(* IEC 61131-3 sources: beebread/doc (part 7) *)

(* ---------------------------------------------- *)
C_SND:
	IF S_BUF.SIZE > 0 THEN
		IF c_ready AND c_enable THEN
			IF NOT s_active THEN
				s_total := LIMIT(0,UINT_TO_INT(S_BUF.SIZE),r_max_size); (* limit and pass total number of bytes *)
				s_cur_pos  := 0;
				s_cur_size := 0;
				s_active := TRUE; (* activate send mode *)
			END_IF;

			s_cur_pos := s_cur_pos + s_cur_size; (* determine new send data position *)
			IF s_total > s_cur_pos THEN (* more data to send? *)
				s_cur_size := s_total - s_cur_pos;
				s_cur_size := LIMIT(0, s_cur_size, s_max_size); (* limit telegram length *)
				s_time := tx; (* reset send timer *)
				r_time := tx; (* reset receive timer *)
				state := C_SND_WAIT1;
			ELSE (* no more send data -> stop sending *)
				s_active := FALSE;
				S_BUF.SIZE := 0;
				state := C_WAIT;
			END_IF;
		END_IF;
	END_IF;

C_SND_WAIT1:
	IF udp_mode THEN
		fbSendTo(bExecute := FALSE );
		fbSendTo(bExecute := TRUE, sSrvNetId := sSrvNetId, hSocket := socket , cbLen := s_cur_size, pSrc := REF(S_BUF.BUFFER[s_cur_pos]), sRemoteHost := s_ip_str, nRemotePort := c_port, tTimeout:= TIME_OUT);
		fbSendTo.bExecute := FALSE;
	ELSE
		fbSend(bExecute := FALSE);
		fbSend(bExecute := TRUE, sSrvNetId := sSrvNetId, hSocket := socket , cbLen:= s_cur_size, pSrc:=REF(S_BUF.BUFFER[s_cur_pos]), tTimeout:= TIME_OUT);
		fbSend.bExecute := FALSE;
	END_IF;
	state := C_SND_WAIT2;

C_SND_WAIT2:
	IF udp_mode THEN
		fbSendTo();
		Send_Busy := fbSendTo.bBusy;
		Send_Error := fbSendTo.bError;
		Send_ErrId := fbSendTo.nErrId;
	ELSE
		fbSend();
		Send_Busy := fbSend.bBusy;
		Send_Error := fbSend.bError;
		Send_ErrId := fbSend.nErrId;
	END_IF;

	IF NOT Send_Busy THEN
		IF NOT Send_Error THEN
    			(*####################  DEBUG-MESSAGE  ###################################*)
			(*########################################################################*)
			state := C_SND;
		ELSE
			nErrId := Send_ErrId;
			state := C_WAIT;
    			(*####################  DEBUG-MESSAGE  ###################################*)
			(*########################################################################*)
		END_IF;
	END_IF;

END_CASE;

(* ---------------------------------------------- *)

IF c_ready THEN
	IF NOT c_ready_old THEN (* connection established - rising edge detected *)
		IP_C.C_STATE := 254;
		IP_C.TIME_RESET := TRUE; (* reset all timers *)
    		(*####################  DEBUG-MESSAGE  ###################################*)
		(*########################################################################*)
	ELSE
		IP_C.C_STATE := 255; (* connection is established *)
	END_IF;
ELSE
	IF c_ready_old THEN (* connection closed - falling edge detected *)
		IP_C.C_STATE := 1;
		IP_C.MAILBOX[1] := 0; (* reset receive info *)
		IP_C.MAILBOX[2] := 0; (* reset send pause *)
		IP_C.MAILBOX[3] := 0; (* reset receive pause *)
		IF NOT new_connection THEN
			s_active := FALSE; (* stop send activities *)
			S_BUF.SIZE := 0; (* clear send length *)
			(*IP_C.TIME_RESET := TRUE; *) (* reset all timers *)
		END_IF;
    		(*####################  DEBUG-MESSAGE  ###################################*)
		(*########################################################################*)

	ELSE
		IP_C.C_STATE := 0; (* connection is closed *)
	END_IF;
END_IF;

c_ready_old := c_ready;

(* ---------------------------------------------- *)

IF IP_C.R_OBSERVE = FALSE OR s_active THEN
    r_time := tx;
END_IF;

IF c_status = 0 AND tx - c_time > error_time AND c_enable AND NOT c_ready AND c_mode < 2 THEN (* Connect Timeout *)
	c_status := 255; (* output timeout error *)
END_IF;
IF s_status = 0 AND tx - s_time > error_time AND s_active THEN (* Send Timeout *)
	s_status := 255; (* output timeout error *)
END_IF;
IF r_status = 0 AND tx - r_time > error_time AND c_ready AND IP_C.R_OBSERVE THEN (* Receive Timeout *)
	r_status := 255; (* output timeout error *)
END_IF;

IP_C.ERROR := DWORD_OF_BYTE(c_status,s_status,r_status,0);

(*####################  DEBUG-MESSAGE  ###################################*)
(*########################################################################*)
END_FUNCTION_BLOCK

FUNCTION_BLOCK IP_CONTROL2
VAR_IN_OUT
	IP_C : IP_C; (* IP_Control management structure *)
	S_BUF : NETWORK_BUFFER_SHORT; (* external send buffer *)
	R_BUF : NETWORK_BUFFER_SHORT; (* external receive buffer *)
END_VAR
VAR_INPUT
	IP : DWORD; (* IP address *)
	PORT : WORD; (* port number *)
	TIME_OUT : TIME; (* monitoring time connect / send / receive *)
END_VAR
VAR
	c_time : UDINT; (* CONNECT time (time without a connection) *)
	s_time : UDINT; (* SEND time    (time since last data sent) *)
	r_time : UDINT; (* RECEIVE time (time since last data received) *)

	c_enable : BOOL; (* Connect: enable *)
	c_ip : DWORD; (* Connect: current IP address *)
	c_ip_str : STRING(15);
	c_port : WORD; (* Connect: current port number *)
	c_mode : BYTE; (* Connect: current mode UDP/TCP...... *)
	c_status : BYTE; (* Connect: Status (Errorcode) *)
	c_ready : BOOL; (* Connect: connection established *)
	c_ready_old : BOOL; (* Connect: last state of c_ready for edge evaluation *)

	s_total : INT; (* Send: total number of bytes to send *)
	s_cur_pos : INT; (* Send: current send position *)
	s_cur_size : INT; (* Send: current send size *)
	s_max_size : INT; (* Send: maximum telegram length for sending *)
	s_active : BOOL; (* Send: data sending is active *)
	s_status : BYTE; (* Send: Status (Errorcodes) *)
	s_ip_str : STRING(15);
	s_ip_exist : BOOL;

	r_status : BYTE; (* Receive: Status (Errorcodes) *)
	r_count : INT; (* Receive: number of received bytes *)
	r_offset : INT; (* Receive: current position in external receive buffer *)
	r_max_size : INT; (* Receive: size of the external receive buffer*)

	new_connection : BOOL; (* new connection parameters available *)
	tx : DWORD; (* last time value *)
	error_time : DWORD; (* current timeout value *)

	state: BYTE; (* step flag for connect *)
	bytes_received : DINT;
	udp_mode : BOOL;

	socket : T_HSOCKET;
	server : T_HSOCKET;
	fbCreate	: FB_SocketUdpCreate;
	fbConnect : FB_SocketConnect;
	fbClose : FB_SocketClose;
	fbSendTo : FB_SocketUdpSendTo;
	fbReceiveFrom : FB_SocketUdpReceiveFrom;
	fbSend : FB_SocketSend;
	fbReceive : FB_SocketReceive;
	fbListen : FB_SocketListen;
	fbAccept : FB_SocketAccept;
	nErrId : UDINT;
	Send_Busy : BOOL;
	Send_Error : BOOL;
	Send_ErrId : UDINT;

	IPCR : IP_CONTROL_RESET;

END_VAR

VAR CONSTANT
	STOP : BYTE := 0;
	UDP_INIT : BYTE:= 31;
	UDP_INIT_WAIT : BYTE:= 32;
	TC_INIT : BYTE := 51;
	TC_CONNECT : BYTE:= 52;
	TS_INIT : BYTE:= 53;
	TS_LISTEN_WAIT : BYTE:= 54;
	TS_ACCEPT : BYTE:= 55;
	TS_ACCEPT_WAIT : BYTE:= 56;
	C_CLOSE : BYTE := 190;
	C_CLOSE_WAIT : BYTE:= 191;
	C_CLOSE2 : BYTE := 192;
	C_CLOSE_WAIT2 : BYTE:= 193;
	C_WAIT : BYTE := 200;
	C_REC : BYTE := 210;
	C_REC_WAIT : BYTE := 211;
	C_SND : BYTE := 220;
	C_SND_WAIT1 : BYTE := 221;
	C_SND_WAIT2 : BYTE := 222;
END_VAR

(* on PLC reset or program download all old connections are closed *)
IPCR();
IF NOT IPCR.READY THEN RETURN; END_IF;

(* ---------------------- Debug-Message ----------------------------*)
(* -----------------------------------------------------------------------------*)

(* read system time *)
tx := T_PLC_MS();

IF IP_C.C_PORT = 0 THEN
	IP_C.C_PORT := PORT; (* replace the given PORT with the configured PORT *)
END_IF;
IF IP_C.C_IP = 0 AND IP_C.C_MODE < 4 THEN
	IP_C.C_IP := IP; (* replace the given IP with the configured IP *)
END_IF;

new_connection := c_ip <> IP_C.C_IP OR c_mode <> IP_C.C_MODE OR c_port <> IP_C.C_PORT; (* new connection requested? *)
c_enable := IP_C.C_ENABLE AND NOT new_connection;

IF IP_C.C_ENABLE AND IP_C.ERROR = 0 AND state = STOP THEN (* enabled, no error, no socket open *)
	c_ip   := IP_C.C_IP;
	c_mode := IP_C.C_MODE;
	c_port := IP_C.C_PORT;
	c_ip_str := IP4_TO_STRING(c_ip);
	udp_mode := C_MODE.0; (* Mode 1,3,5 = udp *)

	error_time := TIME_TO_DWORD(MAX(T#200ms,TIME_OUT));
	IP_C.TIME_RESET := TRUE; (* reset all timers *)
	r_max_size := SIZEOF(R_BUF.BUFFER);
	s_max_size := SIZEOF(S_BUF.BUFFER);

	IF udp_mode THEN (* Mode: 1,3,5 = UDP CLIENT/SERVER *)
		state := UDP_INIT;
	ELSIF c_mode = 0 THEN (* Mode: 0 = TCP CLIENT *)
		state := TC_INIT;
	ELSE
		state := TS_INIT; (* Mode: 2,4 = TCP SERVER *)
	END_IF;

	IF c_mode < 5 THEN (* set receiver IP *)
		s_ip_str := c_ip_str;
		s_ip_exist := TRUE;
	ELSE
		s_ip_str := '';
		s_ip_exist := FALSE;
	END_IF;

	(* ---------------------- Debug-Message ----------------------------*)
	(* -----------------------------------------------------------------------------*)

END_IF;

(* ---------------------- Debug-Message ----------------------------*)
(* -----------------------------------------------------------------------------*)

IF IP_C.TIME_RESET THEN (* reset all timers *)
	IP_C.TIME_RESET := FALSE; (* clear reset *)
	c_time := tx; (* reset connect timer *)
	s_time := tx; (* reset send timer *)
	r_time := tx; (* reset receive timer *)

	c_status := BYTE#0; (* reset last connect error *)
	s_status := BYTE#0; (* reset last send error *)
	r_status := BYTE#0; (* reset last receive error *)
END_IF;

(* ---------------------------------------------- *)

CASE state OF

UDP_INIT: (* UDP_CLIENT + SERVER *)

	fbCreate(bExecute := FALSE);
	fbCreate(	bExecute := TRUE , sSrvNetId := sSrvNetId, sLocalHost := sLocalHost, nLocalPort := SEL(c_mode = 1,c_port,0) , tTimeOut := TIME_OUT);
	fbCreate.bExecute := FALSE; (* presetting *)
	state := UDP_INIT_WAIT;

UDP_INIT_WAIT:
	fbCreate();
	IF NOT fbCreate.bBusy THEN
		IF NOT fbCreate.bError THEN
			socket := fbCreate.hSocket;
			c_ready := TRUE; (* Connected *)
			state := C_WAIT;
		ELSE
			c_status := 1; (* FB_SocketUdpCreate failed *)
			nErrId := fbCreate.nErrId;
			state := C_CLOSE;
		END_IF;
	END_IF;

(* ---------------------------------------------- *)
TC_INIT: (* TCP CLIENT (ACTIVE) *)
	fbConnect(bExecute := FALSE);
	fbConnect(bExecute := TRUE, sSrvNetId := sSrvNetId, sRemoteHost := c_ip_str, nRemotePort := c_port, tTimeout := TIME_OUT);
	fbConnect.bExecute := FALSE; (* presetting *)
	state := TC_CONNECT;

(* ---------------------------------------------- *)
TC_CONNECT:
	IF NOT c_enable OR c_status = 255 THEN (* not enabled or connect timeout *)
		state := C_CLOSE;
	END_IF;

	fbConnect();
	IF NOT fbConnect.bBusy THEN
		IF fbConnect.bError THEN
			nErrID := fbConnect.nErrId;
			state :=TC_INIT; (* try again *)
		ELSE
			socket := fbConnect.hSocket;
			c_ready := TRUE; (* Connected *)
			state := C_WAIT;
		END_IF;
	END_IF;
(* ---------------------------------------------- *)
TS_INIT: (* TCP SERVER (PASSIVE) *)
	fbListen(bExecute := FALSE);
	fbListen(bExecute := TRUE , sSrvNetId:= sSrvNetId , sLocalHost:= sLocalHost , nLocalPort:= c_port , tTimeout:= TIME_OUT);
	fbListen.bExecute := FALSE;
	state := TS_LISTEN_WAIT;
(* ---------------------------------------------- *)
TS_LISTEN_WAIT:
	fbListen();
	IF NOT fbListen.bBusy THEN
		IF fbListen.bError THEN
			c_status := 3; (* FB_SocketListen failed *)
			nErrID := fbListen.nErrId;
			state := C_CLOSE;
		ELSE
			server := fbListen.hListener;
			state := TS_ACCEPT;
		END_IF;
	END_IF;
(* ---------------------------------------------- *)
TS_ACCEPT:
	fbAccept(bExecute := FALSE);
	fbAccept(bExecute := TRUE, sSrvNetId := sSrvNetId, hListener := server, tTimeout := TIME_OUT);
	fbAccept.bExecute := FALSE;
	state := TS_ACCEPT_WAIT;
(* ---------------------------------------------- *)
TS_ACCEPT_WAIT:
	fbAccept();
	IF NOT fbAccept.bBusy THEN

		state := TS_ACCEPT; (* presetting  *)

		IF fbAccept.bError THEN
			c_status := 4; (* FB_SocketAccept failed *)
			nErrID := fbAccept.nErrId;
			state := C_CLOSE;
		ELSE (* no error *)
			IF fbAccept.bAccepted THEN
				socket := fbAccept.hSocket;
				IF socket.remoteAddr.sAddr  <> c_ip_str AND c_mode <> 4 THEN
					state := C_CLOSE; (* reject remote - close connection *)
				ELSE
					state := C_WAIT;
					c_ready := TRUE; (* Connected *)
				END_IF;
			END_IF; (* fbAccept.bAccepted *)
		END_IF; (* NOT fbAccept.bError *)
	END_IF; (*  NOT fbAccept.bBusy *)
(* ---------------------------------------------- *)
C_CLOSE:
	c_ready := FALSE;
	IF socket.handle > 0 THEN
		fbClose(bExecute := FALSE );
		fbClose(bExecute := TRUE, sSrvNetId := sSrvNetId,	hSocket := socket);
		fbClose.bExecute := FALSE;
		state := C_CLOSE_WAIT;
	ELSE
		state:= C_CLOSE2;
	END_IF;

C_CLOSE_WAIT:
	fbClose();
	IF NOT fbClose.bBusy THEN
		socket := TCPADS_NULL_HSOCKET; (* reset socket *)
		nErrId:= SEL(fbClose.bError,0,fbClose.nErrId);
		state:= C_CLOSE2;
	END_IF;

C_CLOSE2:
	IF server.handle > 0 THEN
		fbClose(bExecute := FALSE );
		fbClose(bExecute := TRUE, sSrvNetId := sSrvNetId,	hSocket := server);
		fbClose.bExecute := FALSE;
		state := C_CLOSE_WAIT2;
	ELSE
		state:= STOP;
	END_IF;

C_CLOSE_WAIT2:
	fbClose();
	IF NOT fbClose.bBusy THEN
		server := TCPADS_NULL_HSOCKET; (* reset socket *)
		nErrId:= SEL(fbClose.bError,0,fbClose.nErrId);
		state:= STOP;
	END_IF;

(* ---------------------------------------------- *)

C_WAIT: (* wait for request to close *)
	IF NOT c_enable OR NOT c_ready THEN
		state:= C_CLOSE;
	ELSIF S_BUF.SIZE > 0 AND IP_C.MAILBOX[2] = 0 AND s_ip_exist THEN
		state:= C_SND;
	ELSIF IP_C.MAILBOX[3] = 0 THEN
		state:= C_REC;
	END_IF;

(* ---------------------------------------------- *)

C_REC: (* receive data *)
	IF R_BUF.SIZE >= INT_TO_UINT(r_max_size) THEN
		R_BUF.SIZE := UINT#0;
		r_status := 254; (* receive buffer reset due to overflow *)
	END_IF;

	r_offset := SEL(udp_mode,UINT_TO_INT(R_BUF.SIZE),0);
	r_count := r_max_size - r_offset;
	bytes_received := 0;

	IF udp_mode THEN
		fbReceiveFrom(bExecute := FALSE );
		fbReceiveFrom(bExecute:= TRUE, sSrvNetId := sSrvNetId, hSocket:= socket, cbLen := r_count, pDest:= REF(R_BUF.BUFFER), tTimeout:= TIME_OUT);
		fbReceiveFrom.bExecute := FALSE; (* presetting *)
	ELSE
		fbReceive(bExecute:= FALSE);
		fbReceive(bExecute:= TRUE, sSrvNetId := sSrvNetId , hSocket:= socket , cbLen:= r_count, pDest:= REF(R_BUF.BUFFER[r_offset]) , tTimeout:= TIME_OUT);
		fbReceive.bExecute:= FALSE;
	END_IF;
	state := C_REC_WAIT;

C_REC_WAIT:
	IF udp_mode THEN
		fbReceiveFrom(); (* UDP Mode *)
		IF NOT fbReceiveFrom.bBusy THEN
			IF NOT fbReceiveFrom.bError THEN
				IF fbReceiveFrom.nRecBytes > 0 THEN
					IF c_mode <> BYTE#5 AND fbReceiveFrom.sRemoteHost  <> c_ip_str THEN
						R_BUF.SIZE := UINT#0;
					ELSE
						bytes_received := fbReceiveFrom.nRecBytes;
						IF NOT s_ip_exist THEN
							s_ip_str := fbReceiveFrom.sRemoteHost;
							s_ip_exist := TRUE;
						END_IF;
					END_IF;
				END_IF;
				state := C_WAIT;
			ELSIF fbReceiveFrom.nErrId = 16#80072746 THEN (* connection closed by remote *)
				c_status := 253;
				c_ready := FALSE;
				state := C_WAIT;
			ELSE
				nErrId := fbReceiveFrom.nErrId;
				state := C_WAIT;
			END_IF;
		END_IF;
	ELSE
		fbReceive(); (* TCP Mode *)
		IF NOT fbReceive.bBusy THEN
			IF NOT fbReceive.bError THEN
				IF fbReceive.nRecBytes > 0 THEN
					bytes_received := fbReceive.nRecBytes;
				END_IF;
			ELSIF fbReceive.nErrId = 16#8004 THEN (* connection closed by remote *)
				c_status := 253;
				c_ready := FALSE;
			ELSE
				nErrId := fbReceive.nErrId;
			END_IF;
			state := C_WAIT;
		END_IF;
	END_IF;

	IF bytes_received > 0 THEN
		r_time := tx; (* reset receive timer *)
		R_BUF.SIZE := INT_TO_UINT(r_offset + DINT_TO_UINT(bytes_received)); (* enter current buffer size *)
		IP_C.MAILBOX[1] := IP_C.MAILBOX[1] + 1; (* Receive Info *)
		IF IP_C.MAILBOX[1] = 0 THEN IP_C.MAILBOX[1] := 1; END_IF;
		(* ---------------------- Debug-Message ----------------------------*)
		(* -----------------------------------------------------------------------------*)
	END_IF;

(* ---------------------------------------------- *)
C_SND:
	IF S_BUF.SIZE > 0 THEN
		IF c_ready AND c_enable THEN
			IF NOT s_active THEN
				s_total := LIMIT(0,UINT_TO_INT(S_BUF.SIZE),r_max_size); (* limit and pass total number of bytes *)
				s_cur_pos  := 0;
				s_cur_size := 0;
				s_active := TRUE; (* activate send mode *)
			END_IF;

			s_cur_pos := s_cur_pos + s_cur_size; (* determine new send data position *)
			IF s_total > s_cur_pos THEN (* more data to send? *)
				s_cur_size := s_total - s_cur_pos;
				s_cur_size := LIMIT(0, s_cur_size, s_max_size); (* limit telegram length *)
				s_time := tx; (* reset send timer *)
				r_time := tx; (* reset receive timer *)
				state := C_SND_WAIT1;
			ELSE (* no more send data -> stop sending *)
				s_active := FALSE;
				S_BUF.SIZE := 0;
				state := C_WAIT;
			END_IF;
		END_IF;
	END_IF;

C_SND_WAIT1:
	IF udp_mode THEN
		fbSendTo(bExecute := FALSE );
		fbSendTo(bExecute := TRUE, sSrvNetId := sSrvNetId, hSocket := socket , cbLen := s_cur_size, pSrc := REF(S_BUF.BUFFER[s_cur_pos]), sRemoteHost := s_ip_str, nRemotePort := c_port, tTimeout:= TIME_OUT);
		fbSendTo.bExecute := FALSE;
	ELSE
		fbSend(bExecute := FALSE);
		fbSend(bExecute := TRUE, sSrvNetId := sSrvNetId, hSocket := socket , cbLen:= s_cur_size, pSrc:=REF(S_BUF.BUFFER[s_cur_pos]), tTimeout:= TIME_OUT);
		fbSend.bExecute := FALSE;
	END_IF;
	state := C_SND_WAIT2;

C_SND_WAIT2:
	IF udp_mode THEN
		fbSendTo();
		Send_Busy := fbSendTo.bBusy;
		Send_Error := fbSendTo.bError;
		Send_ErrId := fbSendTo.nErrId;
	ELSE
		fbSend();
		Send_Busy := fbSend.bBusy;
		Send_Error := fbSend.bError;
		Send_ErrId := fbSend.nErrId;
	END_IF;

	IF NOT Send_Busy THEN
		IF NOT Send_Error THEN
			(* ---------------------- Debug-Message ----------------------------*)
			(* -----------------------------------------------------------------------------*)
			state := C_SND;
		ELSE
			nErrId := Send_ErrId;
			state := C_WAIT;
			(* ---------------------- Debug-Message ----------------------------*)
			(* -----------------------------------------------------------------------------*)
		END_IF;
	END_IF;

END_CASE;

(* ---------------------------------------------- *)

IF c_ready THEN
	IF NOT c_ready_old THEN (* connection established - rising edge detected *)
		IP_C.C_STATE := 254;
		IP_C.TIME_RESET := TRUE; (* reset all timers *)
		(* ---------------------- Debug-Message ----------------------------*)
		(* -----------------------------------------------------------------------------*)
	ELSE
		IP_C.C_STATE := 255; (* connection is established *)
	END_IF;
ELSE
	IF c_ready_old THEN (* connection closed - falling edge detected *)
		IP_C.C_STATE := 1;
		IP_C.MAILBOX[1] := 0; (* reset receive info *)
		IP_C.MAILBOX[2] := 0; (* reset send pause *)
		IP_C.MAILBOX[3] := 0; (* reset receive pause *)
		IF NOT new_connection THEN
			s_active := FALSE; (* stop send activities *)
			S_BUF.SIZE := 0; (* clear send length *)
			(* IP_C.TIME_RESET := TRUE; *) (* reset all timers *)
		END_IF;
		(* ---------------------- Debug-Message ----------------------------*)
		(* -----------------------------------------------------------------------------*)

	ELSE
		IP_C.C_STATE := 0; (* connection is closed *)
	END_IF;
END_IF;

c_ready_old := c_ready;

(* ---------------------------------------------- *)

IF IP_C.R_OBSERVE = FALSE OR s_active THEN
    r_time := tx;
END_IF;

IF c_status = 0 AND tx - c_time > error_time AND c_enable AND NOT c_ready AND c_mode < 2 THEN (* Connect Timeout *)
	c_status := 255; (* output timeout error *)
END_IF;
IF s_status = 0 AND tx - s_time > error_time AND s_active THEN (* Send Timeout *)
	s_status := 255; (* output timeout error *)
END_IF;
IF r_status = 0 AND tx - r_time > error_time AND c_ready AND IP_C.R_OBSERVE THEN (* Receive Timeout *)
	r_status := 255; (* output timeout error *)
END_IF;

IP_C.ERROR := DWORD_OF_BYTE(c_status,s_status,r_status,0);

(* ---------------------- Debug-Message ----------------------------*)
(* -----------------------------------------------------------------------------*)
END_FUNCTION_BLOCK

FUNCTION_BLOCK IP_CONTROL_RESET
VAR_INPUT
END_VAR
VAR_OUTPUT
	READY : BOOL;
END_VAR
VAR
	fbSocketCloseAll : FB_SocketCloseAll;
	step : BYTE;
END_VAR
(* On PLC reset or program download close all old connections *)

CASE TCP_SERVER_RESET OF

2:	READY := TRUE;
	RETURN;

1:	IF step = 0 THEN
		RETURN;
	END_IF;

0:	TCP_SERVER_RESET := 1; (* reset is active *)
	step := 1;

END_CASE;

CASE step OF

0:	RETURN;

1:	fbSocketCloseAll(sSrvNetId:= '', bExecute:= TRUE, tTimeout:= T#10s );
	step := 2;

2:	fbSocketCloseAll(bExecute:= FALSE);
	IF fbSocketCloseAll.bBusy = FALSE THEN
		step := 0;
		TCP_SERVER_RESET := 2; (* reset done, ready for use *)
	END_IF;

END_CASE;
END_FUNCTION_BLOCK

FUNCTION_BLOCK IP_FIFO
VAR_IN_OUT
	FIFO : IP_FIFO_DATA;
	ID : BYTE;
	STATE : BYTE;
END_VAR
VAR
	tmp : INT;

END_VAR

IF NOT FIFO.INIT THEN
	FIFO.INIT := TRUE;
	FIFO.NW := 1;
	FIFO.NR := 1;
	FIFO.EMPTY := TRUE;
	FIFO.FULL := FALSE;
	FIFO.TOP := 128; (* array size 1 to x *)
	FIFO.MAX_ID := BYTE#1; (* maximum number of registrations of an ID *)
END_IF;

(* if no ID is present, assign the next free ID *)
IF ID = BYTE#00 THEN
	IF FIFO.ID < INT_TO_BYTE(FIFO.TOP) THEN
		ID := USINT_TO_BYTE(BYTE_TO_USINT(FIFO.ID) + USINT#1); (* ID +1 *)
		FIFO.ID := ID; (* enter ID *)
	    	(*####################  DEBUG-MESSAGE  ###################################*)
	    	(*########################################################################*)
	ELSIF STATE < BYTE#200 THEN
		(*####################  DEBUG-MESSAGE  ###################################*)
		(*########################################################################*)

		(* should never happen! -> too many participants are registered *)
		(* no number is assigned and all requests are answered negatively *)
		STATE := BYTE#255;
		RETURN;
	END_IF;
END_IF;

IF STATE = BYTE#1 AND NOT FIFO.FULL THEN (* register *)
	(* enter only if the maximum number was not exceeded *)
	tmp := BYTE_TO_INT(ID);
	IF FIFO.Y[tmp] < FIFO.MAX_ID THEN
		FIFO.Y[tmp] := USINT_TO_BYTE(BYTE_TO_USINT(FIFO.Y[tmp]) + USINT#1); (* IP_ID counter +1 *)
		tmp := FIFO.NW; (* unfortunately no other way works for me *)
		FIFO.X[tmp] := ID;
		IF FIFO.NW = FIFO.TOP THEN FIFO.NW := 1; ELSE FIFO.NW := FIFO.NW + 1; END_IF;
		FIFO.FULL := FIFO.NW = FIFO.NR;
		FIFO.EMPTY := FALSE;
		STATE := BYTE#2; (* advance to "wait for release" *)
		(*####################  DEBUG-MESSAGE  ###################################*)
		(*########################################################################*)

	END_IF;
END_IF;

IF STATE = BYTE#2 AND NOT FIFO.EMPTY THEN (* check current stack element *)
	tmp := FIFO.NR; (* unfortunately no other way works for me *)
	IF ID = FIFO.X[tmp] THEN
	STATE := BYTE#3; (* advance to "access release" *)
	END_IF;
END_IF;

IF STATE = BYTE#4 AND NOT FIFO.EMPTY THEN (* remove from stack *)
	tmp := FIFO.NR; (* unfortunately no other way works for me *)
	IF ID = FIFO.X[tmp] THEN
		tmp := BYTE_TO_INT(ID); (* unfortunately no other way works for me *)
		FIFO.Y[tmp] := USINT_TO_BYTE(BYTE_TO_USINT(FIFO.Y[tmp]) - USINT#1); (* ID counter -1 *)
		IF FIFO.NR = FIFO.TOP THEN FIFO.NR := 1; ELSE FIFO.NR := FIFO.NR + 1; END_IF;
		FIFO.EMPTY := FIFO.NR = FIFO.NW;
		FIFO.FULL := FALSE;
		(*####################  DEBUG-MESSAGE  ###################################*)
		(*########################################################################*)
	END_IF;
	STATE := BYTE#5; (* "Remove done" *)
END_IF;
END_FUNCTION_BLOCK

// Commented out for beedance: it reads or writes the bytes of a STRING through a pointer; a beedance reference (REF_TO) refers to a whole variable of its type.
// FUNCTION_BLOCK IRTRANS_DECODE
// VAR_IN_OUT
// 	IP_C : IP_C; (* IP_Control management structure *)
// 	R_BUF : NETWORK_BUFFER_SHORT;
// END_VAR
// VAR_OUTPUT
// 	CMD : BOOL;
// 	DEV : STRING;
// 	KEY : STRING;
// 	ERROR : BOOL;
// END_VAR
// VAR
// 	i : INT;
// 	stop : INT;
// 	pt : REF_TO BYTE;
// 	buffer : REF_TO ARRAY[0..32000] OF BYTE;
// 	size : UINT;
// 	z : BYTE;
// END_VAR
//
// size := R_BUF.SIZE;
//
// (* do nothing if the buffer is empty *)
// IF size > 0 AND IP_C.MAILBOX[1] <> z THEN
// 	i := 0;
// 	error := TRUE;
// 	stop := size - 2;
// 	(* read characters before first comma and store in device *)
// 	pt := REF(dev);
// 	buffer := REF(R_BUF.BUFFER);
// 	WHILE i < stop DO
// 		IF buffer^[i] = 44 THEN EXIT; END_IF;
// 		pt^ := buffer^[i];
// 		pt := pt + 1;
// 		i := i + 1;
// 	END_WHILE;
// 	(* terminate the device string *)
// 	pt^ := 0;
// 	(* read after first comma and store in key *)
// 	i := i + 1;
// 	pt := REF(key);
// 	WHILE i < stop DO
// 		pt^ := buffer^[i];
// 		pt := pt + 1;
// 		i := i + 1;
// 	END_WHILE;
// 	(* terminate the key string *)
// 	pt^:= 0;
// 	(* check if last two characters are $R$N 13, 10 *)
// 	IF buffer^[i] <> 13 AND buffer^[i+1] <> 10 THEN	RETURN;	END_IF;
// 	(* check if device and key are present *)
// 	IF LEN(dev) = 0 OR LEN(key) = 0 THEN RETURN; END_IF;
// 	(* a valid transmission has been received *)
// 	cmd := TRUE;
// 	error := FALSE;
// ELSE
// 	error := FALSE;
// 	cmd := FALSE;
// END_IF;
//
// z := IP_C.MAILBOX[1];
// END_FUNCTION_BLOCK

FUNCTION_BLOCK IRTRANS_RCV_1
VAR_INPUT CONSTANT
	DEV_CODE : STRING;
	KEY_CODE : STRING;
END_VAR
VAR_INPUT
	CMD : BOOL;
END_VAR
VAR_IN_OUT
	DEV : STRING;
	KEY : STRING;
END_VAR
VAR_OUTPUT
	Q : BOOL;
END_VAR

Q := cmd AND dev_code = dev AND key_code = key;
END_FUNCTION_BLOCK

FUNCTION_BLOCK IRTRANS_RCV_4
VAR_INPUT CONSTANT
	DEV_CODE : STRING;
	KEY_CODE_0 : STRING;
	KEY_CODE_1 : STRING;
	KEY_CODE_2 : STRING;
	KEY_CODE_3 : STRING;
END_VAR
VAR_INPUT
	CMD : BOOL;
END_VAR
VAR_IN_OUT
	DEV : STRING;
	KEY : STRING;
END_VAR
VAR_OUTPUT
	Q0, Q1, Q2, Q3 : BOOL;
END_VAR
VAR_TEMP
	decode: BOOL;
END_VAR

decode := cmd AND dev_code = dev;

Q0 := key = key_code_0 AND decode;
Q1 := key = key_code_1 AND decode;
Q2 := key = key_code_2 AND decode;
Q3 := key = key_code_3 AND decode;
END_FUNCTION_BLOCK

FUNCTION_BLOCK IRTRANS_RCV_8
VAR_INPUT CONSTANT
	dev_code : STRING;
	key_code_0 : STRING;
	key_code_1 : STRING;
	key_code_2 : STRING;
	key_code_3 : STRING;
	key_code_4 : STRING;
	key_code_5 : STRING;
	key_code_6 : STRING;
	key_code_7 : STRING;
END_VAR
VAR_INPUT
	CMD : BOOL;
END_VAR
VAR_IN_OUT
	DEV : STRING;
	KEY : STRING;
END_VAR
VAR_OUTPUT
	Q0, Q1, Q2, Q3, Q4, Q5, Q6, Q7 : BOOL;
END_VAR
VAR_TEMP
	decode: BOOL;
END_VAR

decode := cmd AND dev_code = dev;

Q0 := key = key_code_0 AND decode;
Q1 := key = key_code_1 AND decode;
Q2 := key = key_code_2 AND decode;
Q3 := key = key_code_3 AND decode;
Q4 := key = key_code_4 AND decode;
Q5 := key = key_code_5 AND decode;
Q6 := key = key_code_6 AND decode;
Q7 := key = key_code_7 AND decode;
END_FUNCTION_BLOCK

FUNCTION_BLOCK IRTRANS_SERVER
VAR_IN_OUT
	IP_C : IP_C; (* IP_Control management structure *)
	S_BUF : NETWORK_BUFFER_SHORT;
	R_BUF : NETWORK_BUFFER_SHORT;
END_VAR
VAR_INPUT
	UDP_TCP : BOOL;
END_VAR
VAR_OUTPUT
	S_ENABLE : BOOL;
	R_ENABLE : BOOL;
	ERROR : DWORD;
END_VAR
VAR
	t : TON;
END_VAR

IF NOT IP_C.C_ENABLE THEN
	(* set up IP data traffic *)
	IP_C.C_PORT := WORD#0; (* enter port number *)
	IP_C.C_IP := DWORD#00; (* enter IP *)
	IP_C.C_MODE := SEL(UDP_TCP,5,4); (* 4 = Mode: TCP+PASSIV+PORT / 5 = Mode: UDP+PASSIV+PORT*)
	IP_C.C_ENABLE := TRUE; (* enable connection setup *)
	IP_C.R_OBSERVE := FALSE; (* monitor data reception *)
	IP_C.TIME_RESET := TRUE; (* reset timeout monitoring *)
	S_BUF.SIZE := UINT#0; (* reset send data *)
	R_BUF.SIZE := UINT#0; (* reset receive data *)
END_IF;

R_ENABLE := IP_C.C_STATE > 127;
S_ENABLE := R_ENABLE AND (IP_C.MAILBOX[1] > 0 OR IP_C.C_MODE <> 5);
ERROR := IP_C.ERROR;

t(IN:= IP_C.ERROR > 0, PT:=T#5s);
IF t.Q THEN
	IP_C.TIME_RESET := TRUE; (* Error Reset *)
END_IF;
END_FUNCTION_BLOCK

// Commented out for beedance: it uses _STRING_TO_BUFFER, which is commented out.
// FUNCTION_BLOCK IRTRANS_SND_1
// VAR_INPUT CONSTANT
// 	DEV_CODE : STRING;
// 	KEY_CODE : STRING;
// END_VAR
// VAR_INPUT
// 	IN : BOOL;
// 	T_REPEAT : TIME;
// END_VAR
// VAR_IN_OUT
// 	IP_C : IP_C; (* IP_Control management structure *)
// 	S_BUF : NETWORK_BUFFER_SHORT;
// END_VAR
// VAR_OUTPUT
// 	KEY : BYTE;
// END_VAR
// VAR
// 	skey : STRING;
// 	size : INT;
// 	str : STRING;
// 	t : TON;
// 	k : BYTE;
// 	lk : BYTE;
// 	d : BOOL;
// END_VAR
//
// d := IP_C.C_STATE > 127 AND (IP_C.MAILBOX[1] > 0 OR IP_C.C_MODE <> 5);
// IF NOT d THEN RETURN; END_IF;
//
// t(IN:= lk = k , PT:=T_REPEAT);
//
// IF S_BUF.SIZE = 0 THEN
// 	IF IN THEN
// 		skey := KEY_CODE; k := 1;
// 	ELSE
// 		lk := 0;
// 		KEY := 0;
// 		RETURN; (* exit if no key is active *)
// 	END_IF;
//
// 	IF lk <> k OR T.Q THEN (* other key or repeat wait time elapsed *)
// 		str := CONCAT('snd ',dev_code);
// 		str := CONCAT(str,',');
// 		str := CONCAT(str,skey);
// 		size := LEN(str);
// 		_STRING_TO_BUFFER(STR:=str, POS:=0, PT:=REF(S_BUF.BUFFER), SIZE:=size);
// 		S_BUF.SIZE := size; (* enter send length *)
// 		KEY := k;
// 		lk := k; (* store last key *)
// 		t(IN:=FALSE); (* Reset Time *)
// 	END_IF;
// END_IF;
// END_FUNCTION_BLOCK

// Commented out for beedance: it uses _STRING_TO_BUFFER, which is commented out.
// FUNCTION_BLOCK IRTRANS_SND_4
// VAR_INPUT CONSTANT
// 	DEV_CODE : STRING;
// 	KEY_CODE_0 : STRING;
// 	KEY_CODE_1 : STRING;
// 	KEY_CODE_2 : STRING;
// 	KEY_CODE_3 : STRING;
// END_VAR
// VAR_INPUT
// 	IN_0 : BOOL;
// 	IN_1 : BOOL;
// 	IN_2 : BOOL;
// 	IN_3 : BOOL;
// 	T_REPEAT : TIME;
// END_VAR
// VAR_IN_OUT
// 	IP_C : IP_C; (* IP_Control management structure *)
// 	S_BUF : NETWORK_BUFFER_SHORT;
// END_VAR
// VAR_OUTPUT
// 	KEY : BYTE;
// END_VAR
// VAR
// 	skey : STRING;
// 	size : INT;
// 	str : STRING;
// 	t : TON;
// 	k : BYTE;
// 	lk : BYTE;
// 	d : BOOL;
// END_VAR
//
// d := IP_C.C_STATE > 127 AND (IP_C.MAILBOX[1] > 0 OR IP_C.C_MODE <> 5);
// IF NOT d THEN RETURN; END_IF;
//
// t(IN:= lk = k , PT:=T_REPEAT);
//
// IF S_BUF.SIZE = 0 THEN
// 	IF IN_0 THEN
// 		skey := KEY_CODE_0; k := 1;
// 	ELSIF IN_1 THEN
// 		skey := KEY_CODE_1; k := 2;
// 	ELSIF IN_2 THEN
// 		skey := KEY_CODE_2; k := 3;
// 	ELSIF IN_3 THEN
// 		skey := KEY_CODE_3; k := 4;
// 	ELSE
// 		lk := 0;
// 		KEY := 0;
// 		RETURN; (* exit if no key is active *)
// 	END_IF;
//
// 	IF lk <> k OR T.Q THEN (* other key or repeat wait time elapsed *)
// 		str := CONCAT('snd ',dev_code);
// 		str := CONCAT(str,',');
// 		str := CONCAT(str,skey);
// 		size := LEN(str);
// 		_STRING_TO_BUFFER(STR:=str, POS:=0, PT:=REF(S_BUF.BUFFER), SIZE:=size);
// 		S_BUF.SIZE := size; (* enter send length *)
// 		KEY := k;
// 		lk := k; (* store last key *)
// 		t(IN:=FALSE); (* Reset Time *)
// 	END_IF;
// END_IF;
// END_FUNCTION_BLOCK

// Commented out for beedance: it uses _STRING_TO_BUFFER, which is commented out.
// FUNCTION_BLOCK IRTRANS_SND_8
// VAR_INPUT CONSTANT
// 	DEV_CODE : STRING;
// 	KEY_CODE_0 : STRING;
// 	KEY_CODE_1 : STRING;
// 	KEY_CODE_2 : STRING;
// 	KEY_CODE_3 : STRING;
// 	KEY_CODE_4 : STRING;
// 	KEY_CODE_5 : STRING;
// 	KEY_CODE_6 : STRING;
// 	KEY_CODE_7 : STRING;
// END_VAR
// VAR_INPUT
// 	IN_0 : BOOL;
// 	IN_1 : BOOL;
// 	IN_2 : BOOL;
// 	IN_3 : BOOL;
// 	IN_4 : BOOL;
// 	IN_5 : BOOL;
// 	IN_6 : BOOL;
// 	IN_7 : BOOL;
// 	T_REPEAT : TIME;
// END_VAR
// VAR_IN_OUT
// 	IP_C : IP_C; (* IP_Control management structure *)
// 	S_BUF : NETWORK_BUFFER_SHORT;
// END_VAR
// VAR_OUTPUT
// 	KEY : BYTE;
// END_VAR
// VAR
// 	skey : STRING;
// 	size : INT;
// 	str : STRING;
// 	t : TON;
// 	k : BYTE;
// 	lk : BYTE;
// 	d : BOOL;
// END_VAR
//
// d := IP_C.C_STATE > 127 AND (IP_C.MAILBOX[1] > 0 OR IP_C.C_MODE <> 5);
// IF NOT d THEN RETURN; END_IF;
//
// t(IN:= lk = k , PT:=T_REPEAT);
//
// IF S_BUF.SIZE = 0 THEN
// 	IF IN_0 THEN
// 		skey := KEY_CODE_0; k := 1;
// 	ELSIF IN_1 THEN
// 		skey := KEY_CODE_1; k := 2;
// 	ELSIF IN_2 THEN
// 		skey := KEY_CODE_2; k := 3;
// 	ELSIF IN_3 THEN
// 		skey := KEY_CODE_3; k := 4;
// 	ELSIF IN_4 THEN
// 		skey := KEY_CODE_4; k := 5;
// 	ELSIF IN_5 THEN
// 		skey := KEY_CODE_5; k := 6;
// 	ELSIF IN_6 THEN
// 		skey := KEY_CODE_6; k := 7;
// 	ELSIF IN_7 THEN
// 		skey := KEY_CODE_7; k := 8;
// 	ELSE
// 		lk := 0;
// 		KEY := 0;
// 		RETURN; (* exit if no key is active *)
// 	END_IF;
//
// 	IF lk <> k OR T.Q THEN (* other key or repeat wait time elapsed *)
// 		str := CONCAT('snd ',dev_code);
// 		str := CONCAT(str,',');
// 		str := CONCAT(str,skey);
// 		size := LEN(str);
// 		_STRING_TO_BUFFER(STR:=str, POS:=0, PT:=REF(S_BUF.BUFFER), SIZE:=size);
// 		S_BUF.SIZE := size; (* enter send length *)
// 		KEY := k;
// 		lk := k; (* store last key *)
// 		t(IN:=FALSE); (* Reset Time *)
// 	END_IF;
// END_IF;
// END_FUNCTION_BLOCK

// Commented out for beedance: it uses COUNT_CHAR, which is commented out.
// FUNCTION IS_IP4 : BOOL
// VAR_INPUT
// 	str : STRING;
// END_VAR
//
// IS_IP4 := COUNT_CHAR(str, 46) = 3;
// END_FUNCTION

FUNCTION IS_URLCHR : BOOL
VAR_INPUT
	IN : BYTE;
END_VAR

IS_URLCHR := ((IN > 47) AND (IN < 58)) OR ((IN > 64) AND (IN < 91)) OR ((IN > 96) AND (IN < 123)) OR (in = 126) OR (in = 95) OR (in =45) OR (in =46);
END_FUNCTION

// Commented out for beedance: it uses PRINT_SF, which is commented out.
// FUNCTION_BLOCK LOG_MSG
// (* VAR_EXTERNAL
// 	LOG_CL :	LOG_CONTROL;
// END_VAR *)
// VAR
// 	FB_PRINT_SF :PRINT_SF;
// 	idX : INT;
// END_VAR
//
// IF DWORD_TO_BYTE(SHL(LOG_CL.NEW_MSG_OPTION,16)) > LOG_CL.LEVEL THEN RETURN; END_IF; (* logging enabled?*)
//
// FB_PRINT_SF(PRINTF_DATA := LOG_CL.PRINTF,STR := LOG_CL.NEW_MSG);
//
// IF LOG_CL.RESET THEN (* delete log entries *)
// 	LOG_CL.RESET := FALSE;
// 	LOG_CL.RING_MODE := FALSE;
// 	LOG_CL.IDX := 0;
// 	LOG_CL.UPDATE_COUNT := LOG_CL.UPDATE_COUNT + UINT#1; (* increment UpdateCount *)
// END_IF;
//
// IF LOG_CL.SIZE > 0 THEN (* size value is entered *)
// 	IF LEN(LOG_CL.NEW_MSG) > 0 THEN (* enter message into buffer *)
// 		IF (LOG_CL.IDX >= LOG_CL.SIZE) THEN
// 			LOG_CL.RING_MODE := TRUE; (* on overflow = ring buffer mode *)
// 			LOG_CL.IDX := 0; (* position at start of array again *)
// 		END_IF;
//
// 		LOG_CL.UPDATE_COUNT := LOG_CL.UPDATE_COUNT + UINT#1; (* increment UpdateCount *)
// 		LOG_CL.IDX := LOG_CL.IDX + INT#1; (* next free position *)
// 		idx := LOG_CL.IDX; (* load current log buffer position *)
// 		LOG_CL.MSG[idx] := LOG_CL.NEW_MSG; (* store new log string in buffer  *)
// 		LOG_CL.MSG_OPTION[idx] := LOG_CL.NEW_MSG_OPTION; (* store new log string option in buffer  *)
// 		LOG_CL.NEW_MSG := ''; (* delete last log string *)
// 	END_IF;
// END_IF;
// END_FUNCTION_BLOCK

FUNCTION_BLOCK LOG_VIEWPORT
VAR_IN_OUT
	LC : LOG_CONTROL;
	LV : us_LOG_VIEWPORT;
END_VAR
VAR
	pos : INT;
	count : INT;
	idx : INT;
	base : INT;
	update_pos : BOOL;
END_VAR

(* process scroll button *)
IF LV.MOVE_TO_X <> 0 THEN
	CASE LV.MOVE_TO_X OF
	30000: pos := 1 ; (* show oldest message *)
	30001: pos := LC.SIZE; (* show newest message *)
	30002: pos := pos + LV.COUNT; (* page down -> towards newer messages *)
	30003: pos := pos - LV.COUNT; (* page up -> towards older messages *)
	ELSE
		pos := pos + LV.MOVE_TO_X;
	END_CASE;
	update_pos := TRUE;
	LV.MOVE_TO_X := 0;
END_IF;

IF (LV.UPDATE_COUNT <> LC.UPDATE_COUNT) OR update_pos THEN (* monitor update *)
	LV.UPDATE := TRUE;
	LV.UPDATE_COUNT := LC.UPDATE_COUNT;
	update_pos := FALSE;

	(* check and take pos *)
	IF LC.RING_MODE THEN
		pos := LIMIT(1,pos,LC.SIZE - LV.COUNT + 1);
	ELSE
		IF LC.IDX > LV.COUNT THEN
			pos := LIMIT(1,pos,LC.IDX - LV.COUNT + 1);
		ELSE
			pos := 1;
		END_IF;
	END_IF;

	(* calculate idxBasis *)
	base := LC.IDX - pos - LV.COUNT + 1;
	IF LC.RING_MODE THEN
		(* display in ring buffer mode *)
		FOR count:= 1 TO LV.COUNT DO
			idx := base + count;
			IF idx < 1 THEN
				idx := idx + LC.SIZE;
			END_IF;
			LV.LINE_ARRAY[count] := idx;
		END_FOR;
	ELSE
		(* display in normal mode *)
		FOR count:= 1 TO LV.COUNT DO
			idx := base + count;
			IF idx < 1 THEN
				(* output empty line *)
				LV.LINE_ARRAY[count] := 0;
			ELSE
				LV.LINE_ARRAY[count] := idx;
			END_IF;
		END_FOR;
	END_IF;
END_IF;
END_FUNCTION_BLOCK

FUNCTION_BLOCK MB_CLIENT
VAR_IN_OUT
	IP_C : IP_C;
	S_BUF : NETWORK_BUFFER_SHORT;
	R_BUF : NETWORK_BUFFER_SHORT;
	DATA : ARRAY [0..255] OF WORD;
END_VAR
VAR_INPUT
	DATA_SIZE : INT;
	ENABLE : BOOL;
	UDP : BOOL;
	FC : INT;
	UNIT_ID : BYTE;
	R_ADDR : INT;
	R_POINTS : INT;
	R_DATA_ADR : INT;
	R_DATA_BITPOS : INT;
	W_ADDR : INT;
	W_POINTS : INT;
	W_DATA_ADR : INT;
	W_DATA_BITPOS : INT;
	DELAY : TIME;
END_VAR
VAR_OUTPUT
	ERROR : DWORD;
	BUSY : BOOL;
END_VAR
VAR
	ip_state : BYTE;
	ip_id : BYTE;
	ip_fifo : ip_fifo;
	mask : DWORD;
	w_tmp : WORD;
	idx1 : INT;
	idx2 : INT;
	stop : INT;
	i : INT;
	bit_pos : INT;
	w_mask : WORD;
	b_mask : BYTE;
	count : INT;
	state : INT;
	transaction_id : INT;
	response : INT;
	comp : INT;
	ton_1 : TON;
END_VAR

CASE state OF

00: (* wait for delay time *)
	TON_1(IN:=ENABLE,PT:=DELAY);

	IF TON_1.Q OR DELAY = T#0s THEN
		TON_1(IN:=FALSE);
		state := 20;
		IP_STATE := BYTE#1; (* register *)
	END_IF;

20: (* register with IP_Control *)
	IF IP_STATE = BYTE#3 THEN
		(* set up IP data traffic *)
		IP_C.C_PORT := WORD#0; (* use port from IP_CONTROL *)
		IP_C.C_IP := DWORD#0; (* use IP from IP_CONTROL *)
		IP_C.C_MODE := BOOL_TO_BYTE(UDP); (* Mode: 0=TCP+ACTIVE+IP , 1=UDP+ACTIVE+IP *)
		IP_C.TIME_RESET := TRUE; (* reset timeout monitoring *)
		IP_C.C_ENABLE := TRUE; (* enable connection setup *)
		IP_C.R_OBSERVE := TRUE; (* receive monitoring *)
		ERROR := DWORD#00; (* reset last error *)

		(******************************************************************)
		CASE FC OF
		1..2: (* 0x01 Read Coil Status , 0x02 Read Input Status *)
			IF R_POINTS <= 2000 THEN
				w_tmp := INT_TO_WORD(R_ADDR);
				S_BUF.BUFFER[08] := WORD_TO_BYTE(SHR(w_tmp,8));
				S_BUF.BUFFER[09] := WORD_TO_BYTE(w_tmp);
				w_tmp := INT_TO_WORD(R_POINTS);
				S_BUF.BUFFER[10] := WORD_TO_BYTE(SHR(w_tmp,8));
				S_BUF.BUFFER[11] := WORD_TO_BYTE(w_tmp);
				S_BUF.SIZE := UINT#12;
				Response :=	WORD_TO_INT(SHR(INT_TO_WORD(R_POINTS + 7),3));
				comp := 7;
			ELSE
				ERROR := DWORD#2; (* ILLEGAL DATA ADDRESS *)
			END_IF;
		(******************************************************************)
		3..4: (* 0x03 Read Holding Registers , 0x04 Read Input Registers *)
			IF R_POINTS <= 125 THEN
				w_tmp := INT_TO_WORD(R_ADDR);
				S_BUF.BUFFER[08] := WORD_TO_BYTE(SHR(w_tmp,8));
				S_BUF.BUFFER[09] := WORD_TO_BYTE(w_tmp);
				w_tmp := INT_TO_WORD(R_POINTS);
				S_BUF.BUFFER[10] := WORD_TO_BYTE(SHR(w_tmp,8));
				S_BUF.BUFFER[11] := WORD_TO_BYTE(w_tmp);
				S_BUF.SIZE := UINT#12;
				Response :=	WORD_TO_INT(SHL(w_tmp,1));
				comp := 7;
			ELSE
				ERROR := DWORD#2; (* ILLEGAL DATA ADDRESS *)
			END_IF;
		(******************************************************************)
		5:	(* 0x05 Force Single Coil *)
			IF W_DATA_ADR <= DATA_SIZE THEN
				w_tmp := INT_TO_WORD(W_ADDR);
				S_BUF.BUFFER[08] := WORD_TO_BYTE(SHR(w_tmp,8));
				S_BUF.BUFFER[09] := WORD_TO_BYTE(w_tmp);
				S_BUF.BUFFER[10] := SEL((DATA[W_DATA_ADR] AND SHL(WORD#1,W_DATA_BITPOS))>WORD#00,BYTE#16#00,BYTE#16#FF);
				S_BUF.BUFFER[11] := BYTE#00;
				S_BUF.SIZE := UINT#12;
				Response := 3;
				comp := 11;
			ELSE
				ERROR := DWORD#2; (* ILLEGAL DATA ADDRESS *)
			END_IF;
		(******************************************************************)
		6:	(* 0x06 Preset Single Register *)
			IF W_DATA_ADR <= DATA_SIZE THEN
				w_tmp := INT_TO_WORD(W_ADDR);
				S_BUF.BUFFER[08] := WORD_TO_BYTE(SHR(w_tmp,8));
				S_BUF.BUFFER[09] := WORD_TO_BYTE(w_tmp);
				w_tmp := DATA[W_DATA_ADR];
				S_BUF.BUFFER[10] := WORD_TO_BYTE(SHR(w_tmp,8));
				S_BUF.BUFFER[11] := WORD_TO_BYTE(w_tmp);
				S_BUF.SIZE := UINT#12;
				Response := 3;
				comp := 11;
			ELSE
				ERROR := DWORD#2; (* ILLEGAL DATA ADDRESS *)
			END_IF;
		(******************************************************************)
		15:	(* 0x0F Force Multiple Coils *)
			IF (WORD_TO_INT(SHR(INT_TO_WORD(WORD_TO_INT(SHL(INT_TO_WORD(W_DATA_ADR),4)) + W_POINTS + W_DATA_BITPOS + 15),4)) <= DATA_SIZE) AND W_POINTS <= 1968 THEN
				w_tmp := INT_TO_WORD(W_ADDR);
				S_BUF.BUFFER[08] := WORD_TO_BYTE(SHR(w_tmp,8));
				S_BUF.BUFFER[09] := WORD_TO_BYTE(w_tmp);
				w_tmp := INT_TO_WORD(W_POINTS);
				S_BUF.BUFFER[10] := WORD_TO_BYTE(SHR(w_tmp,8));
				S_BUF.BUFFER[11] := WORD_TO_BYTE(w_tmp);
				S_BUF.BUFFER[12] := WORD_TO_BYTE(SHR(INT_TO_WORD(W_POINTS + 7),3));

				w_mask := SHL(WORD#1,W_DATA_BITPOS);
				bit_pos := 0;
				w_tmp := WORD#00;
				idx1 := 12;
				idx2 := W_DATA_ADR;
				FOR i := 1 TO W_POINTS DO
					w_tmp :=BIT_LOAD_W(w_tmp,(DATA[idx2] AND w_mask) > WORD#0,bit_pos);
					bit_pos := bit_pos + 1;
					IF bit_pos > 7 OR i=W_POINTS THEN
						bit_pos := 0;
						idx1 := idx1 + 1;
						S_BUF.BUFFER[idx1] := WORD_TO_BYTE(w_tmp);
						w_tmp := WORD#0;
					END_IF;
					w_mask := ROL(w_mask,1);
					IF w_mask = WORD#1 THEN
						idx2 := idx2 +1;
					END_IF;
				END_FOR;
				S_BUF.SIZE := INT_TO_UINT(idx1 + 1);
				Response := 3;
				comp := 11;
			ELSE
				ERROR := DWORD#2; (* ILLEGAL DATA ADDRESS *)
			END_IF;
		(******************************************************************)
		16:	(* 0x10 Write Multiple Registers *)
			IF W_DATA_ADR + W_POINTS <= DATA_SIZE AND W_POINTS <= 123 THEN
				w_tmp := INT_TO_WORD(W_ADDR);
				S_BUF.BUFFER[08] := WORD_TO_BYTE(SHR(w_tmp,8));
				S_BUF.BUFFER[09] := WORD_TO_BYTE(w_tmp);
				w_tmp := INT_TO_WORD(W_POINTS);
				S_BUF.BUFFER[10] := WORD_TO_BYTE(SHR(w_tmp,8));
				S_BUF.BUFFER[11] := WORD_TO_BYTE(w_tmp);
				S_BUF.BUFFER[12] := SHL(S_BUF.BUFFER[11],1);

				idx1 := 11;
				count := W_DATA_ADR + W_POINTS - 1;
				FOR i := W_DATA_ADR TO count DO
					idx1 := idx1 + 2;
					idx2 := idx1 + 1; (* second index necessary for pcworx! *)
					w_tmp := DATA[i];
					S_BUF.BUFFER[idx1] := WORD_TO_BYTE(SHR(w_tmp,8));
					S_BUF.BUFFER[idx2] := WORD_TO_BYTE(w_tmp);
				END_FOR;

				S_BUF.SIZE := INT_TO_UINT(idx2 + 1);
				Response := 3;
				comp := 11;
			ELSE
				ERROR := DWORD#2; (* ILLEGAL DATA ADDRESS *)
			END_IF;
		(******************************************************************)
		22:	(* 0x16 Mask Write Register *)
			IF W_DATA_ADR + 2 <= DATA_SIZE THEN
				w_tmp := INT_TO_WORD(W_ADDR);
				S_BUF.BUFFER[08] := WORD_TO_BYTE(SHR(w_tmp,8));
				S_BUF.BUFFER[09] := WORD_TO_BYTE(w_tmp);
				idx1 := W_DATA_ADR;
				w_tmp := DATA[idx1];
				S_BUF.BUFFER[10] := WORD_TO_BYTE(SHR(w_tmp,8));
				S_BUF.BUFFER[11] := WORD_TO_BYTE(w_tmp);
				idx1 := idx1 +1;
				w_tmp := DATA[idx1];
				S_BUF.BUFFER[12] := WORD_TO_BYTE(SHR(w_tmp,8));
				S_BUF.BUFFER[13] := WORD_TO_BYTE(w_tmp);

				S_BUF.SIZE := UINT#14;
				Response := 5;
				comp := 13;
			ELSE
				ERROR := DWORD#2; (* ILLEGAL DATA ADDRESS *)
			END_IF;
		(******************************************************************)
		23:	(* 0x17 Read/Write Multible Registers *)
			IF W_DATA_ADR + W_POINTS <= DATA_SIZE AND W_POINTS <= 121 AND R_POINTS <= 125 THEN
				idx1 := 15;
				count := W_DATA_ADR + W_POINTS - 1;
				FOR i := W_DATA_ADR TO count DO
					idx1 := idx1 + 2;
					idx2 := idx1 + 1; (* second index necessary for pcworx! *)
					w_tmp := DATA[i];
					S_BUF.BUFFER[idx1] := WORD_TO_BYTE(SHR(w_tmp,8));
					S_BUF.BUFFER[idx2] := WORD_TO_BYTE(w_tmp);
				END_FOR;

				(* WRITE *)
				w_tmp := INT_TO_WORD(W_ADDR);
				S_BUF.BUFFER[12] := WORD_TO_BYTE(SHR(w_tmp,8));
				S_BUF.BUFFER[13] := WORD_TO_BYTE(w_tmp);
				w_tmp := INT_TO_WORD(W_POINTS);
				S_BUF.BUFFER[14] := WORD_TO_BYTE(SHR(w_tmp,8));
				S_BUF.BUFFER[15] := WORD_TO_BYTE(w_tmp);
				S_BUF.BUFFER[16] := SHL(S_BUF.BUFFER[15],1);

				(* READ *)
				w_tmp := INT_TO_WORD(R_ADDR);
				S_BUF.BUFFER[08] := WORD_TO_BYTE(SHR(w_tmp,8));
				S_BUF.BUFFER[09] := WORD_TO_BYTE(w_tmp);
				w_tmp := INT_TO_WORD(R_POINTS);
				S_BUF.BUFFER[10] := WORD_TO_BYTE(SHR(w_tmp,8));
				S_BUF.BUFFER[11] := WORD_TO_BYTE(w_tmp);

				S_BUF.SIZE := INT_TO_UINT(idx2 + 1);
				Response := WORD_TO_INT(SHL(w_tmp,1));
				comp := 7;
			ELSE
				ERROR := DWORD#2; (* ILLEGAL DATA ADDRESS *)
			END_IF;
		(******************************************************************)

		ELSE
			ERROR := DWORD#00000001; (* ILLEGAL FUNCTION *)
		END_CASE;

		(* send data *)
		IF ERROR = DWORD#00 THEN
			Transaction_ID := Transaction_ID + 1;
			w_tmp := UINT_TO_WORD(S_BUF.SIZE - UINT#6);
			(* ---- H E A D E R --------------------------------------------------------------- *)
			S_BUF.BUFFER[0] := IP_ID; (* TRANSACTION-ID HI-Byte *)
			S_BUF.BUFFER[1] := INT_TO_BYTE(Transaction_ID); (* TRANSACTION-ID LO-Byte *)
			S_BUF.BUFFER[2] := BYTE#00; (* PROTOCOL ID HI byte *)
			S_BUF.BUFFER[3] := BYTE#00; (* PROTOCOL ID LO byte *)
			S_BUF.BUFFER[4] := WORD_TO_BYTE(SHR(w_tmp,8)); (* length HI byte *)
			S_BUF.BUFFER[5] := WORD_TO_BYTE(w_tmp); (* length LO byte *)
			S_BUF.BUFFER[6] := UNIT_ID; (* UNIT *)
			S_BUF.BUFFER[7] := INT_TO_BYTE(FC); (* FUNCTION-CODE *)
			(*----- END OF HEADER --------------------------------------------------------------*)
			R_BUF.SIZE := UINT#0; (* clear receive buffer *)
			state := 30; (* wait for response *)
		ELSE
			IP_STATE := BYTE#4; (* unregister *)
			state := 00;
		END_IF;
	END_IF;

30: (* response *)
	IF IP_C.ERROR <> DWORD#00 THEN
		ERROR := IP_C.ERROR;
		IP_STATE := BYTE#4; (* unregister *)
		state := 00;
	ELSIF S_BUF.SIZE = UINT#0 AND R_BUF.SIZE > UINT#0 THEN
		(* enter expected length into send buffer afterwards to allow comparison *)
		w_tmp := INT_TO_WORD(Response + 3);
		S_BUF.BUFFER[4] := WORD_TO_BYTE(SHR(w_tmp,8));
		S_BUF.BUFFER[5] := WORD_TO_BYTE(w_tmp);

		FOR i := 0 TO comp DO
			IF S_BUF.BUFFER[i] <> R_BUF.BUFFER[i] THEN EXIT; END_IF;
		END_FOR;

		IF R_BUF.SIZE >= UINT#9 AND R_BUF.BUFFER[7] > BYTE#128 THEN  (* Bit 7 = Error Message *)
			ERROR := BYTE_TO_DWORD(R_BUF.BUFFER[8]);
			IP_STATE := BYTE#4; (* unregister *)
			state := 00;
		ELSIF R_BUF.SIZE = INT_TO_UINT(Response + 9) AND i > comp THEN
			mask := SHL(DWORD#1,FC);
			(* READ_COILS, READ_INPUT_DISCRETES *)
			IF (mask AND DWORD#2#00000000_00000000_00000000_00000110) > DWORD#0 THEN (* FC 1,2 *)
				IF WORD_TO_INT(SHR(INT_TO_WORD(WORD_TO_INT(SHL(INT_TO_WORD(R_DATA_ADR),4)) + R_POINTS + R_DATA_BITPOS + 15),4)) <= DATA_SIZE THEN
					b_mask := BYTE#1;
					idx1 := 09;
					idx2 := R_DATA_ADR;
					bit_pos := R_DATA_BITPOS;
					FOR i := 1 TO R_POINTS DO
						DATA[idx2]:=BIT_LOAD_W(DATA[idx2],(R_BUF.BUFFER[idx1] AND b_mask) > BYTE#0,bit_pos);
						bit_pos := bit_pos + 1;
						IF bit_pos > 15 THEN
							idx2 := idx2 + 1;
							bit_pos := 0;
						END_IF;
						b_mask := ROL(b_mask,1);
						IF b_mask = BYTE#1 THEN
							idx1 := idx1 + 1;
						END_IF;
					END_FOR;
				ELSE
					ERROR := DWORD#2; (* ILLEGAL DATA ADDRESS *)
				END_IF;

			(* READ_MULTIPLE_REGISTERS, READ_INPUT_REGISTERS, READ_WRITE_REGISTERS *)
			ELSIF (mask AND DWORD#2#00000000_10000000_00000000_00011000) > DWORD#0 THEN (* FC 3,4,23 *)
				IF R_DATA_ADR + R_POINTS <= DATA_SIZE THEN
					stop := R_DATA_ADR + R_POINTS -1 ;
					idx1 := 07;
					FOR i := R_DATA_ADR TO stop DO
						idx1 := idx1 + 2;
						idx2 := idx1 + 1;
						DATA[i] := WORD_OF_BYTE(R_BUF.BUFFER[idx1],R_BUF.BUFFER[idx2]);
					END_FOR;
				ELSE
					ERROR := DWORD#2; (* ILLEGAL DATA ADDRESS *)
				END_IF;
			ELSIF (mask AND DWORD#2#11111111_00111110_01111111_10000001) > DWORD#0 THEN (* ILLEGAL FUNCTION CODE ? *)
				ERROR := DWORD#1; (* ILLEGAL FUNCTION *)
			END_IF;
		ELSE
			ERROR := DWORD#3; (* ILLEGAL DATA VALUE *)
		END_IF;

		IP_STATE := BYTE#4; (* unregister *)
		state := 00;
		R_BUF.SIZE := UINT#0;

	END_IF;

END_CASE;

(* IP_FIFO *)
IP_FIFO(FIFO:=IP_C.FIFO,STATE:=IP_STATE,ID:=IP_ID);
BUSY := IP_STATE = BYTE#3;
END_FUNCTION_BLOCK

FUNCTION_BLOCK MB_SERVER
VAR_IN_OUT
	IP_C : IP_C;
	S_BUF : NETWORK_BUFFER_SHORT;
	R_BUF : NETWORK_BUFFER_SHORT;
	VMAP : ARRAY [1..10] OF VMAP_DATA;
	DATA : ARRAY [0..255] OF WORD;
END_VAR
VAR_INPUT
	DATA_SIZE : INT;
	ENABLE : BOOL;
	UDP : BOOL;
END_VAR
VAR_OUTPUT
	ERROR : DWORD;
END_VAR
VAR
	MB_VMAP : MB_VMAP;
	adr1 : INT;
	adr2 : INT;
	points : INT;
	points2 : INT;
	coils : BYTE;
	mask : BYTE;
	idx1 : INT;
	idx2 : INT;
	bit_pos : INT;
	count : INT;
	fc : INT;
	i : INT;
	state : INT;
	ip_state : BYTE;
	ip_id : BYTE;
	IP_FIFO : IP_FIFO;
	w_tmp : WORD;
	last_cycle : TIME;
	tx : TIME;
	t : TON;
	ip_error : BOOL;
END_VAR

(* read system time *)
tx := DWORD_TO_TIME(T_PLC_MS());

FOR i := 1 TO 10 DO
	IF VMAP[i].TIME_OUT > T#0s THEN
		VMAP[i].TIME_OUT := VMAP[i].TIME_OUT + tx - last_cycle;
	END_IF;
END_FOR;
last_cycle := tx;
ip_error := IP_C.ERROR > DWORD#0;

CASE state OF
00: (* wait for release *)
	IF ENABLE THEN
		state := 10;
		ip_state := BYTE#1; (* register *)
	END_IF;

10: (* register with IP_Control and wait for release *)
	IF ip_state = BYTE#3 THEN

		(* set up IP data traffic *)
		IP_C.C_PORT := WORD#0; (* use port from IP_CONTROL *)
		IP_C.C_IP := DWORD#0; (* use IP from IP_CONTROL *)
		IP_C.C_MODE := SEL(UDP,BYTE#4,BYTE#5); (* Mode: 4=TCP+PASSIV+PORT , 5=UDP+PASSIV+PORT *)
		IP_C.TIME_RESET := TRUE; (* reset timeout monitoring *)
		IP_C.C_ENABLE := TRUE; (* enable connection setup *)
		IP_C.R_OBSERVE := TRUE; (* no receive monitoring *)
		state := 20;
	END_IF;

20:	IF NOT ip_error THEN
		IF S_BUF.SIZE = UINT#0 AND R_BUF.SIZE > UINT#6 THEN	(* data sending not active and data was received *)
			IF  R_BUF.SIZE = WORD_TO_UINT(WORD_OF_BYTE(R_BUF.BUFFER[4],R_BUF.BUFFER[5])) + UINT#6 THEN (* valid data length *)
				ERROR := DWORD#00; (* clear error *)

				(* copy header *)
				FOR i := 0 TO 13 DO
					S_BUF.BUFFER[i] := R_BUF.BUFFER[i];
				END_FOR;
				fc := BYTE_TO_INT(R_BUF.BUFFER[7]);
				adr1 := WORD_TO_INT(WORD_OF_BYTE(R_BUF.BUFFER[8],R_BUF.BUFFER[9]));
				points := WORD_TO_INT(WORD_OF_BYTE(R_BUF.BUFFER[10],R_BUF.BUFFER[11]));

				(* Virtual Address *)
				MB_VMAP(VMAP:=VMAP,FC:=fc,V_ADR:=adr1,V_CNT:=points,SIZE:=DATA_SIZE);
				adr1:=MB_VMAP.P_ADR;
				bit_pos:=MB_VMAP.P_BIT;
				ERROR:=BYTE_TO_DWORD(MB_VMAP.ERROR);

				IF ERROR = DWORD#0 THEN
					(*---------------------------------------------*)
					CASE fc OF
					1..2 : (* Read Coil Status / Read Input Status *)
						count := 9; (* first data byte *)
						coils := BYTE#0;
						mask := BYTE#1;
						FOR i := 1 TO points DO
							IF mask = BYTE#0 THEN
								mask := BYTE#1;
								S_BUF.BUFFER[count] := coils;
								coils := BYTE#0;
								count := count + 1;
							END_IF;
							IF (DATA[adr1] AND SHL(WORD#1,bit_pos)) > WORD#0 THEN
								coils := coils OR mask;
							END_IF;

							bit_Pos := bit_Pos + 1;
							IF bit_pos > 15 THEN
								ADR1 := ADR1 + 1;
								bit_pos := 0;
							END_IF;

							mask := SHL(mask,1);
						END_FOR;
						S_BUF.BUFFER[Count] := coils;

						S_BUF.BUFFER[8] := INT_TO_BYTE(count - 8); (* Bytecount *)
						S_BUF.SIZE := INT_TO_UINT(count + 1);

					(*--------------------------------------------------*)
					3..4 : (* Read Holding Registers / Read Input Registers *)
						idx1 := 07;
						count := adr1 + points - 1;
						FOR i := adr1 TO count DO
							idx1 := idx1 + 2;
							idx2 := idx1 + 1; (* second index necessary for pcworx! *)
							w_tmp := DATA[i];
							S_BUF.BUFFER[idx1] := WORD_TO_BYTE(SHR(w_tmp,8));
							S_BUF.BUFFER[idx2] := WORD_TO_BYTE(w_tmp);
						END_FOR;
						S_BUF.BUFFER[8] := SHL(INT_TO_BYTE(points),1); (* number of registers in bytes *)
						S_BUF.SIZE := INT_TO_UINT(idx2 + 1);
					(*--------------------------------------------------*)
					5 : (* Force Single Coil *)
						DATA[adr1]:=BIT_LOAD_W(DATA[adr1],R_BUF.BUFFER[10] > BYTE#0,bit_pos);
						S_BUF.SIZE := UINT#12;
					(*--------------------------------------------------*)
					6 : (* Preset Single Register *)
						DATA[adr1] := WORD_OF_BYTE(R_BUF.BUFFER[10],R_BUF.BUFFER[11]);
						S_BUF.SIZE := UINT#12;
					(*--------------------------------------------------*)
					15 : (* Force Multible Coils *)
						mask := BYTE#1;
						idx1 := 13;
						FOR i := 1 TO points DO
							DATA[adr1]:=BIT_LOAD_W(DATA[adr1],(R_BUF.BUFFER[idx1] AND mask) > BYTE#0,bit_pos);
							bit_pos := bit_pos + 1;
							IF bit_pos > 15 THEN
								adr1:= adr1 + 1;
								bit_pos := 0;
							END_IF;
							mask := ROL(mask,1);
							IF mask = BYTE#1 THEN
								idx1 := idx1 +1;
							END_IF;
						END_FOR;
						S_BUF.SIZE := UINT#12;
					(*--------------------------------------------------*)
					16 : (* Preset Multiple Registers	*)
						idx1 := 11;
						count := adr1 + points - 1;
						FOR i := adr1 TO Count DO
							idx1 := idx1 + 2;
	 						idx2 := idx1 + 1;
							Data[i] := WORD_OF_BYTE(R_BUF.BUFFER[idx1],R_BUF.BUFFER[idx2]);
						END_FOR;
						S_BUF.SIZE := UINT#12;
					(*--------------------------------------------------*)
					22 : (* Mask Write Register *)
						w_tmp := WORD_OF_BYTE(R_BUF.BUFFER[10],R_BUF.BUFFER[11]); (* and mask *)
						DATA[adr1] := (DATA[adr1] AND w_tmp) OR (WORD_OF_BYTE(R_BUF.BUFFER[12],R_BUF.BUFFER[13]) AND (NOT w_tmp));
						S_BUF.SIZE := UINT#14;
					(*--------------------------------------------------*)
					23 : (* Read / Write Registers	*)
						(*--- Write-Register -----------------------------------*)
						adr2 := WORD_TO_INT(WORD_OF_BYTE(R_BUF.BUFFER[12],R_BUF.BUFFER[13]));
						points2 := WORD_TO_INT(WORD_OF_BYTE(R_BUF.BUFFER[14],R_BUF.BUFFER[15]));

						(* Virtual Address Write Register *)
						MB_VMAP(VMAP:=VMAP,FC:=16,V_ADR:=adr2,V_CNT:=points2,SIZE:=DATA_SIZE);
						adr2:=MB_VMAP.P_ADR;
						ERROR:=BYTE_TO_DWORD(MB_VMAP.ERROR);

						IF ERROR = DWORD#0 THEN
							idx1 := 15;
							count := adr2 + points2 - 1;
							FOR i := adr2 TO count DO
								idx1 := idx1 + 2;
	 							idx2 := idx1 + 1; (* second index necessary for pcworx! *)
								Data[i] := WORD_OF_BYTE(R_BUF.BUFFER[idx1],R_BUF.BUFFER[idx2]);
							END_FOR;

							(*--- Read-Register -----------------------------------*)
							idx1 := 07;
							count := adr1 + points - 1;
							FOR i := adr1 TO count DO
								idx1 := idx1 + 2;
								idx2 := idx1 + 1; (* second index necessary for pcworx! *)
								w_tmp := DATA[i];
								S_BUF.BUFFER[idx1] := WORD_TO_BYTE(SHR(w_tmp,8));
								S_BUF.BUFFER[idx2] := WORD_TO_BYTE(w_tmp);
							END_FOR;
							S_BUF.BUFFER[8] := SHL(INT_TO_BYTE(points),1); (* number of registers in bytes *)
							S_BUF.SIZE := INT_TO_UINT(idx2 + 1);

						END_IF;

					(*--------------------------------------------------*)
					ELSE
						ERROR := DWORD#01; (* ILLEGAL FUNCTION *)
					END_CASE;
				END_IF;
			END_IF;

			IF ERROR > DWORD#0 THEN
				S_BUF.BUFFER[7] := S_BUF.BUFFER[7] OR BYTE#2#1000_0000; (* set error bit *)
				S_BUF.BUFFER[8] := DWORD_TO_BYTE(ERROR);
				S_BUF.SIZE := UINT#9;
			END_IF;

			S_BUF.BUFFER[4] := BYTE#0; (* high Byte *)
			S_BUF.BUFFER[5] := UINT_TO_BYTE(S_BUF.SIZE - UINT#6); (* enter length field - low byte only *)

		END_IF;
	ELSE
		ERROR := IP_C.ERROR;
	END_IF;

	t(IN:= ip_error, PT:=T#2s);
	IF t.Q THEN
		IP_C.TIME_RESET := TRUE; (* Error Reset *)
	END_IF;

	R_BUF.SIZE := UINT#0; (* destroy receive data *)

	IF ENABLE = FALSE OR t.Q THEN
	    ip_state := BYTE#4; (* unregister *)
		state := 00;
		IP_C.C_ENABLE := FALSE;
	END_IF;
END_CASE;

(* IP_FIFO *)
IP_FIFO(FIFO:=IP_C.FIFO,STATE:=ip_state,ID:=ip_id);
END_FUNCTION_BLOCK

FUNCTION_BLOCK MB_SERVER_1
VAR_IN_OUT
	IP_C : IP_C;
	S_BUF : NETWORK_BUFFER_SHORT;
	R_BUF : NETWORK_BUFFER_SHORT;
	VMAP : ARRAY [1..10] OF VMAP_DATA;
	DATA : ARRAY [0..255] OF WORD;
END_VAR
VAR_INPUT
	DATA_SIZE : INT;
	ENABLE : BOOL;
	UDP : BOOL;
END_VAR
VAR_OUTPUT
	ERROR : DWORD;
END_VAR
VAR
	MB_VMAP : MB_VMAP;
	adr1 : INT;
	adr2 : INT;
	points : INT;
	points2 : INT;
	coils : BYTE;
	mask : BYTE;
	idx1 : INT;
	idx2 : INT;
	bit_pos : INT;
	count : INT;
	fc : INT;
	i : INT;
	state : INT;
	ip_state : BYTE;
	ip_id : BYTE;
	IP_FIFO : IP_FIFO;
	w_tmp : WORD;
	last_cycle : TIME;
	tx : TIME;
	t : TON;
	ip_error : BOOL;
END_VAR

(* read system time *)
tx := DWORD_TO_TIME(T_PLC_MS());

FOR i := 1 TO 10 DO
	IF VMAP[i].TIME_OUT > T#0s THEN
		VMAP[i].TIME_OUT := VMAP[i].TIME_OUT + tx - last_cycle;
	END_IF;
END_FOR;
last_cycle := tx;
ip_error := IP_C.ERROR > DWORD#0;

CASE state OF
00: (* wait for release *)
	IF ENABLE THEN
		state := 10;
		ip_state := BYTE#1; (* register *)
	END_IF;

10: (* register with IP_Control and wait for release *)
	IF ip_state = BYTE#3 THEN

		(* set up IP data traffic *)
		IP_C.C_PORT := WORD#0; (* use port from IP_CONTROL *)
		IP_C.C_IP := DWORD#0; (* use IP from IP_CONTROL *)
		IP_C.C_MODE := SEL(UDP,BYTE#4,BYTE#5); (* Mode: 4=TCP+PASSIV+PORT , 5=UDP+PASSIV+PORT *)
		IP_C.TIME_RESET := TRUE; (* reset timeout monitoring *)
		IP_C.C_ENABLE := TRUE; (* enable connection setup *)
		IP_C.R_OBSERVE := FALSE; (* no receive monitoring *)
		state := 20;
	END_IF;

20:	IF NOT ip_error THEN
		IF S_BUF.SIZE = UINT#0 AND R_BUF.SIZE > UINT#6 THEN	(* data sending not active and data was received *)
			IF  R_BUF.SIZE = WORD_TO_UINT(WORD_OF_BYTE(R_BUF.BUFFER[4],R_BUF.BUFFER[5])) + UINT#6 THEN (* valid data length *)
				ERROR := DWORD#00; (* clear error *)

				(* copy header *)
				FOR i := 0 TO 13 DO
					S_BUF.BUFFER[i] := R_BUF.BUFFER[i];
				END_FOR;
				fc := BYTE_TO_INT(R_BUF.BUFFER[7]);
				adr1 := WORD_TO_INT(WORD_OF_BYTE(R_BUF.BUFFER[8],R_BUF.BUFFER[9]));
				points := WORD_TO_INT(WORD_OF_BYTE(R_BUF.BUFFER[10],R_BUF.BUFFER[11]));

				(* Virtual Address *)
				MB_VMAP(VMAP:=VMAP,FC:=fc,V_ADR:=adr1,V_CNT:=points,SIZE:=DATA_SIZE);
				adr1:=MB_VMAP.P_ADR;
				bit_pos:=MB_VMAP.P_BIT;
				ERROR:=BYTE_TO_DWORD(MB_VMAP.ERROR);

				IF ERROR = DWORD#0 THEN
					(*---------------------------------------------*)
					CASE fc OF
					1..2 : (* Read Coil Status / Read Input Status *)
						count := 9; (* first data byte *)
						coils := BYTE#0;
						mask := BYTE#1;
						FOR i := 1 TO points DO
							IF mask = BYTE#0 THEN
								mask := BYTE#1;
								S_BUF.BUFFER[count] := coils;
								coils := BYTE#0;
								count := count + 1;
							END_IF;
							IF (DATA[adr1] AND SHL(WORD#1,bit_pos)) > WORD#0 THEN
								coils := coils OR mask;
							END_IF;

							bit_Pos := bit_Pos + 1;
							IF bit_pos > 15 THEN
								ADR1 := ADR1 + 1;
								bit_pos := 0;
							END_IF;

							mask := SHL(mask,1);
						END_FOR;
						S_BUF.BUFFER[Count] := coils;

						S_BUF.BUFFER[8] := INT_TO_BYTE(count - 8); (* Bytecount *)
						S_BUF.SIZE := INT_TO_UINT(count + 1);

					(*--------------------------------------------------*)
					3..4 : (* Read Holding Registers / Read Input Registers *)
						idx1 := 07;
						count := adr1 + points - 1;
						FOR i := adr1 TO count DO
							idx1 := idx1 + 2;
							idx2 := idx1 + 1; (* second index necessary for pcworx! *)
							w_tmp := DATA[i];
							S_BUF.BUFFER[idx1] := WORD_TO_BYTE(SHR(w_tmp,8));
							S_BUF.BUFFER[idx2] := WORD_TO_BYTE(w_tmp);
						END_FOR;
						S_BUF.BUFFER[8] := SHL(INT_TO_BYTE(points),1); (* number of registers in bytes *)
						S_BUF.SIZE := INT_TO_UINT(idx2 + 1);
					(*--------------------------------------------------*)
					5 : (* Force Single Coil *)
						DATA[adr1]:=BIT_LOAD_W(DATA[adr1],R_BUF.BUFFER[10] > BYTE#0,bit_pos);
						S_BUF.SIZE := UINT#12;
					(*--------------------------------------------------*)
					6 : (* Preset Single Register *)
						DATA[adr1] := WORD_OF_BYTE(R_BUF.BUFFER[10],R_BUF.BUFFER[11]);
						S_BUF.SIZE := UINT#12;
					(*--------------------------------------------------*)
					15 : (* Force Multible Coils *)
						mask := BYTE#1;
						idx1 := 13;
						FOR i := 1 TO points DO
							DATA[adr1]:=BIT_LOAD_W(DATA[adr1],(R_BUF.BUFFER[idx1] AND mask) > BYTE#0,bit_pos);
							bit_pos := bit_pos + 1;
							IF bit_pos > 15 THEN
								adr1:= adr1 + 1;
								bit_pos := 0;
							END_IF;
							mask := ROL(mask,1);
							IF mask = BYTE#1 THEN
								idx1 := idx1 +1;
							END_IF;
						END_FOR;
						S_BUF.SIZE := UINT#12;
					(*--------------------------------------------------*)
					16 : (* Preset Multiple Registers	*)
						idx1 := 11;
						count := adr1 + points - 1;
						FOR i := adr1 TO Count DO
							idx1 := idx1 + 2;
	 						idx2 := idx1 + 1;
							Data[i] := WORD_OF_BYTE(R_BUF.BUFFER[idx1],R_BUF.BUFFER[idx2]);
						END_FOR;
						S_BUF.SIZE := UINT#12;
					(*--------------------------------------------------*)
					22 : (* Mask Write Register *)
						w_tmp := WORD_OF_BYTE(R_BUF.BUFFER[10],R_BUF.BUFFER[11]); (* and mask *)
						DATA[adr1] := (DATA[adr1] AND w_tmp) OR (WORD_OF_BYTE(R_BUF.BUFFER[12],R_BUF.BUFFER[13]) AND (NOT w_tmp));
						S_BUF.SIZE := UINT#14;
					(*--------------------------------------------------*)
					23 : (* Read / Write Registers	*)
						(*--- Write-Register -----------------------------------*)
						adr2 := WORD_TO_INT(WORD_OF_BYTE(R_BUF.BUFFER[12],R_BUF.BUFFER[13]));
						points2 := WORD_TO_INT(WORD_OF_BYTE(R_BUF.BUFFER[14],R_BUF.BUFFER[15]));

						(* Virtual Address Write Register *)
						MB_VMAP(VMAP:=VMAP,FC:=16,V_ADR:=adr2,V_CNT:=points2,SIZE:=DATA_SIZE);
						adr2:=MB_VMAP.P_ADR;
						ERROR:=BYTE_TO_DWORD(MB_VMAP.ERROR);

						IF ERROR = DWORD#0 THEN
							idx1 := 15;
							count := adr2 + points2 - 1;
							FOR i := adr2 TO count DO
								idx1 := idx1 + 2;
	 							idx2 := idx1 + 1; (* second index necessary for pcworx! *)
								Data[i] := WORD_OF_BYTE(R_BUF.BUFFER[idx1],R_BUF.BUFFER[idx2]);
							END_FOR;

							(*--- Read-Register -----------------------------------*)
							idx1 := 07;
							count := adr1 + points - 1;
							FOR i := adr1 TO count DO
								idx1 := idx1 + 2;
								idx2 := idx1 + 1; (* second index necessary for pcworx! *)
								w_tmp := DATA[i];
								S_BUF.BUFFER[idx1] := WORD_TO_BYTE(SHR(w_tmp,8));
								S_BUF.BUFFER[idx2] := WORD_TO_BYTE(w_tmp);
							END_FOR;
							S_BUF.BUFFER[8] := SHL(INT_TO_BYTE(points),1); (* number of registers in bytes *)
							S_BUF.SIZE := INT_TO_UINT(idx2 + 1);

						END_IF;

					(*--------------------------------------------------*)
					ELSE
						ERROR := DWORD#01; (* ILLEGAL FUNCTION *)
					END_CASE;
				END_IF;
			END_IF;

			IF ERROR > DWORD#0 THEN
				S_BUF.BUFFER[7] := S_BUF.BUFFER[7] OR BYTE#2#1000_0000; (* set error bit *)
				S_BUF.BUFFER[8] := DWORD_TO_BYTE(ERROR);
				S_BUF.SIZE := UINT#9;
			END_IF;

			S_BUF.BUFFER[4] := BYTE#0; (* high Byte *)
			S_BUF.BUFFER[5] := UINT_TO_BYTE(S_BUF.SIZE - UINT#6); (* enter length field - low byte only *)

		END_IF;
	ELSE
		ERROR := IP_C.ERROR;
	END_IF;

	t(IN:= ip_error, PT:=T#5s);
	IF t.Q THEN
		IP_C.TIME_RESET := TRUE; (* Error Reset *)
	END_IF;

	R_BUF.SIZE := UINT#0; (* destroy receive data *)

	IF ENABLE = FALSE THEN
	    ip_state := BYTE#4; (* unregister *)
		state := 00;
	END_IF;
END_CASE;

(* IP_FIFO *)
IP_FIFO(FIFO:=IP_C.FIFO,STATE:=ip_state,ID:=ip_id);
END_FUNCTION_BLOCK

FUNCTION_BLOCK MB_VMAP
VAR_IN_OUT
	VMAP :  ARRAY [1..10] OF VMAP_DATA;
END_VAR
VAR_INPUT
	FC : INT;
	V_ADR : INT;
	V_CNT : INT;
	SIZE : INT;
END_VAR
VAR_OUTPUT
	P_ADR : INT;
	P_BIT : INT;
	ERROR : BYTE;
END_VAR
VAR
	i : INT;
	vopt : DWORD;
	vadr : INT;
	padr : INT;
	mask : DWORD;
	vsize : INT;
	w_tmp : WORD;
	i_tmp : INT;
	init : BOOL;
END_VAR

IF init = FALSE THEN
	init := TRUE;
	IF VMAP[1].FC = DWORD#0 THEN
		VMAP[1].FC := DWORD#16#FFFF_FFFF;
		VMAP[1].V_ADR := 0;
		VMAP[1].V_SIZE := 256;
		VMAP[1].P_ADR := 0;
	END_IF;
END_IF;

ERROR := BYTE#02; (* ILLEGAL DATA ADDRESS *)
mask := SHL(DWORD#1,FC);

IF (mask AND DWORD#2#00000000_01000000_00000000_01100000) <> DWORD#0 THEN (* FC 5,6,22 *)
	V_CNT := 1;
ELSIF V_CNT = 0 THEN
	RETURN;
END_IF;

FOR i := 1 TO 10 DO
	vopt := VMAP[i].FC;
	IF (vopt AND mask) <> DWORD#0 THEN
		vadr := VMAP[i].V_ADR;
		vsize := VMAP[i].V_SIZE;
		padr := VMAP[i].P_ADR;

		IF (mask AND DWORD#2#00000000_00000000_10000000_00100110) <> DWORD#0 THEN (* FC 1,2,5,15 for bit access *)
			i_tmp := WORD_TO_INT(SHR(INT_TO_WORD(V_ADR + V_CNT -1),4))+1;
			IF i_tmp <= SIZE AND i_tmp <= vsize THEN
				w_tmp := INT_TO_WORD(V_ADR);
				P_ADR := WORD_TO_INT(SHR(w_tmp,4)) + padr;
				P_BIT := WORD_TO_INT(w_tmp AND WORD#16#000F);
				ERROR := BYTE#0;
				EXIT;
			END_IF;
		ELSIF (mask AND DWORD#2#00000000_11000001_00000000_01011000) <> DWORD#0 THEN (* FC 3,4,6,16,22,23 for register access *)
			IF V_ADR >= vadr AND V_ADR + V_CNT <= vadr + vsize THEN (* valid virtual range *)
				P_ADR := V_ADR - vadr + padr; (* calculate real address *)
				IF P_ADR + V_CNT <= SIZE THEN (* out of range? *)
					ERROR := BYTE#0;
					EXIT;
				END_IF;
			END_IF;
		ELSE
			ERROR := BYTE#01; (* ILLEGAL FUNCTION *)
			RETURN;
		END_IF;
	END_IF;
END_FOR;

IF ERROR = BYTE#0 THEN
	IF (mask AND DWORD#2#00000000_11000001_10000000_01100000) <> DWORD#0 THEN (* FC 5,6,15,16,22,23 write access *)
		VMAP[i].TIME_OUT := T#1ms;
	END_IF;
END_IF;
END_FUNCTION_BLOCK

FUNCTION MD5_AUX : DWORD
VAR_INPUT
	N : INT;
	A : DWORD;
	B : DWORD;
	C : DWORD;
	D : DWORD;
	X : DWORD;
	U : INT;
	T : DWORD;
END_VAR
VAR
	w : DWORD;
END_VAR

CASE N OF
	1: w := (B AND C) OR (NOT(B) AND D);
	2: w := (B AND D) OR (C AND NOT D);
	3: w := (B XOR C XOR D);
	4: w := (C XOR (B OR  NOT(D)));
END_CASE

MD5_AUX := B + ROL(A + w + X + T,U);
END_FUNCTION

// Commented out for beedance: it uses MD5_TO_STRH, which is commented out.
// FUNCTION_BLOCK MD5_CRAM_AUTH
// VAR_IN_OUT
// 	RUN : BOOL;
// 	USERNAME : STRING(64);
// 	PASSWORD : STRING(64);
// 	B64_TS : STRING(64);  (* Base64 coded ServerTimeStamp *)
// 	AUTH_KEY : STRING(192);
// END_VAR
// VAR
// 	BASE64_DECODE_STR : BASE64_DECODE_STR;
// 	BASE64_ENCODE_STR : BASE64_ENCODE_STR;
// 	MD5_STREAM : MD5_STREAM;
// 	step : INT;
// 	md5_mode : INT;
// 	buf : ARRAY [0..63] OF BYTE;
// 	md5 : ARRAY [0..15] OF BYTE;
// 	md5_first : ARRAY [0..15] OF BYTE;
// 	md5_str1 : STRING(64);
// 	md5_str2 : STRING(64);
// 	size : UDINT;
// 	n1 : INT;
// 	n2 : INT;
// 	pos : UDINT;
// 	b64d_run : BOOL;
// 	b64d_done : BOOL;
// 	b64e_run : BOOL;
// 	b64e_done : BOOL;
// 	str_192 : STRING(192);
// 	str_144 : STRING(144);
// 	xpad : BYTE;
// 	pt : REF_TO BYTE;
// END_VAR
//
// CASE step OF
//
// 0:	IF RUN THEN
// 		step := 5;
// 		str_192 := B64_TS;
// 		b64d_run := TRUE;
// 	END_IF;
//
// 5: IF B64D_DONE THEN (* IPAD cycle *)
// 		b64d_run := FALSE;
// 		xpad := 16#36;
// 		md5_str1 := PASSWORD;
// 		md5_str2 := str_144;
// 		size := 64 + LEN(md5_str2);
// 		md5_mode := 1;
// 		step := 10;
// 	END_IF;
//
// 10: IF md5_mode = 3 THEN (* OPAD Zyklus *)
// 		md5_first := md5; (* save md5 array of IPAD *)
// 		xpad := 16#5C;
// 		size := 64 + 16;
// 		md5_mode := 1;
// 		step := 20;
// 	END_IF;
//
// 20: IF md5_mode = 3 THEN
// 		md5_mode := 0;
// 		str_144 := CONCAT(USERNAME , ' ');
// 		str_144 := CONCAT(str_144 , MD5_TO_STRH(md5));
// 		b64e_run := TRUE;
// 		step := 30;
// 	END_IF;
//
// 30: IF B64E_DONE THEN
// 		AUTH_KEY := str_192;
// 		b64e_run := FALSE;
// 		RUN := FALSE;
// 		step := 0; (* all finished !! *)
// 	END_IF;
//
// END_CASE;
//
// (* ----------- md5 -------------- *)
// CASE md5_mode OF
//
// 1:	n2 := LEN(md5_str1) - 1;
// 	pt := REF(md5_str1);
// 	FOR n1 := 0 TO n2 DO (* copy string into buf *)
// 		buf[n1] := pt^ XOR xpad;
// 		pt := pt + 1;
// 	END_FOR;
// 	FOR n1 := n2 + 1 TO 63 DO (* fill with ipad *)
// 		buf[n1] := xpad;
// 	END_FOR;
//
// 2:	(* Data copy and Calc *)
// 	IF size > 0 AND pos >= 64 THEN
// 		IF step = 20 THEN
// 			FOR n1 := 0 TO 15 DO
// 				buf[n1] := md5_first[n1];
// 			END_FOR;
// 		ELSE
// 			n2 := LEN(md5_str2) - 1;
// 			pt := REF(md5_str2);
// 			FOR n1 := 0 TO n2 DO (* copy string into buf *)
// 				buf[n1] := pt^;
// 				pt := pt + 1;
// 			END_FOR;
// 		END_IF;
// 	END_IF;
//
// END_CASE;
//
// IF md5_mode > 0 THEN
// 	MD5_STREAM(SIZE:=size, MODE:=md5_mode, BUF:=buf, MD5:=md5, POS=>pos);
// END_IF;
//
// BASE64_DECODE_STR(RUN:=b64d_run, STR1:=str_192, STR2:=str_144, DONE=>b64d_done);
// BASE64_ENCODE_STR(RUN:=b64e_run, STR1:=str_144, STR2:=str_192, DONE=>b64e_done);
// END_FUNCTION_BLOCK

// Commented out for beedance: it uses _STRING_TO_BUFFER, which is commented out.
// FUNCTION_BLOCK MD5_STR
// VAR_INPUT
// 	RUN: BOOL;
// END_VAR
// VAR_OUTPUT
// 	DONE: BOOL;
// END_VAR
// VAR_IN_OUT
// 	STR: STRING(STRING_LENGTH);
// 	MD5 : ARRAY [0..15] OF BYTE;
// END_VAR
// VAR
// 	run_last: BOOL;
// 	MD5_STREAM : MD5_STREAM;
// 	buf : ARRAY [0..63] OF BYTE;
// 	mode : INT;
// 	size : UDINT;
// 	pos : UDINT;
// END_VAR
//
// CASE mode OF
// 0:	(* wait for start *)
// 	IF RUN AND NOT run_last THEN
// 		DONE := FALSE;
// 		mode := 1; (* initialization *)
// 		size := LEN(STR);
// 	END_IF;
//
// 2:	(* Data copy and Calc *)
// 	IF size > 0 THEN
// 		_STRING_TO_BUFFER(STR:=MID(STR, UDINT_TO_INT(SIZE), UDINT_TO_INT(POS) + 1), POS:=0, PT:=REF(buf), SIZE:=SIZEOF(buf));
// 	END_IF;
//
// 3:	DONE := TRUE;
// 	mode := 0; (* Stop *)
//
// END_CASE;
//
// IF mode > 0 THEN
// 	MD5_STREAM(SIZE:=size, MODE:=mode, BUF:=buf, MD5:=MD5, POS=>pos);
// END_IF;
//
// run_last := RUN;
// END_FUNCTION_BLOCK

FUNCTION_BLOCK MD5_STREAM
VAR_IN_OUT
	MODE : INT;
	BUF : ARRAY [0..63] OF BYTE;
	MD5 : ARRAY [0..15] OF BYTE;
	SIZE : UDINT;
END_VAR

VAR_OUTPUT
	POS : UDINT;
END_VAR

VAR
	hash : ARRAY [0..3] OF DWORD;
	a : DWORD;
	b : DWORD;
	c : DWORD;
	d : DWORD;
	end : UDINT;
	block : UDINT;
	x : ARRAY [0..15] OF DWORD;
	n : INT;
	n1 : INT;
	z : INT;
	pad_1 : BOOL;
END_VAR

CASE MODE OF

1:	(* initialization of the hash values *)
	hash[0] := DWORD#16#67452301;
	hash[1] := DWORD#16#EFCDAB89;
	hash[2] := DWORD#16#98BADCFE;
	hash[3] := DWORD#16#10325476;

	block := SHR(SIZE,6) + BOOL_TO_UDINT((UDINT_TO_BYTE(SIZE) AND 16#3F) > 55);
	pad_1 := FALSE;
	POS := 0;
	End := SIZE;
	SIZE := MIN(64,End);
	MODE := 2;

2:	(* append padding bytes *)
	FOR n := UDINT_TO_INT(SIZE) TO 63 DO
		BUF[n] := 0;
	END_FOR;

	IF SIZE < 64 AND NOT pad_1 THEN
		BUF[SIZE] := 2#1000_0000;
		pad_1 := TRUE;
	END_IF;

	POS := POS + SIZE;
	SIZE := MIN(64,End - POS);

	n := 0;	(* copy byte array into DWORD array *)
	FOR n1 := 0 TO 15 DO
		x[n1] := DWORD_OF_BYTE(BUF[n+3],BUF[n+2],BUF[n+1],BUF[n]); (* Little Endian Format *)
		n := n + 4;
	END_FOR;

	IF block = 0 THEN (* enter the data length at the end of the last block *)
		x[14] := SHL(UDINT_TO_DWORD(End),3); (* enter number of data bits in little-endian format *)
		MODE := 3;
	ELSE
		block := block - 1;
	END_IF;

	a := hash[0];
	b := hash[1];
	c := hash[2];
	d := hash[3];

	a := MD5_AUX(1, a, b, c, d, X[00], 07, 16#D76AA478); (* 01 *)
	d := MD5_AUX(1, d, a, b, c, X[01], 12, 16#E8C7B756); (* 02 *)
	c := MD5_AUX(1, c, d, a, b, X[02], 17, 16#242070DB); (* 03 *)
	b := MD5_AUX(1, b, c, d, a, X[03], 22, 16#C1BDCEEE); (* 04 *)
	a := MD5_AUX(1, a, b, c, d, X[04], 07, 16#F57C0FAF); (* 05 *)
	d := MD5_AUX(1, d, a, b, c, X[05], 12, 16#4787C62A); (* 06 *)
	c := MD5_AUX(1, c, d, a, b, X[06], 17, 16#A8304613); (* 07 *)
	b := MD5_AUX(1, b, c, d, a, X[07], 22, 16#FD469501); (* 08 *)
	a := MD5_AUX(1, a, b, c, d, X[08], 07, 16#698098D8); (* 09 *)
	d := MD5_AUX(1, d, a, b, c, X[09], 12, 16#8B44F7AF); (* 10 *)
	c := MD5_AUX(1, c, d, a, b, X[10], 17, 16#FFFF5BB1); (* 11 *)
	b := MD5_AUX(1, b, c, d, a, X[11], 22, 16#895CD7BE); (* 12 *)
	a := MD5_AUX(1, a, b, c, d, X[12], 07, 16#6B901122); (* 13 *)
	d := MD5_AUX(1, d, a, b, c, X[13], 12, 16#FD987193); (* 14 *)
	c := MD5_AUX(1, c, d, a, b, X[14], 17, 16#A679438E); (* 15 *)
	b := MD5_AUX(1, b, c, d, a, X[15], 22, 16#49B40821); (* 16 *)

	a := MD5_AUX(2, a, b, c, d, X[01], 05, 16#F61E2562); (* 17 *)
	d := MD5_AUX(2, d, a, b, c, X[06], 09, 16#C040B340); (* 18 *)
	c := MD5_AUX(2, c, d, a, b, X[11], 14, 16#265E5A51); (* 19 *)
	b := MD5_AUX(2, b, c, d, a, X[00], 20, 16#E9B6C7AA); (* 20 *)
	a := MD5_AUX(2, a, b, c, d, X[05], 05, 16#D62F105D); (* 21 *)
	d := MD5_AUX(2, d, a, b, c, X[10], 09, 16#02441453); (* 22 *)
	c := MD5_AUX(2, c, d, a, b, X[15], 14, 16#D8A1E681); (* 23 *)
	b := MD5_AUX(2, b, c, d, a, X[04], 20, 16#E7D3FBC8); (* 24 *)
	a := MD5_AUX(2, a, b, c, d, X[09], 05, 16#21E1CDE6); (* 25 *)
	d := MD5_AUX(2, d, a, b, c, X[14], 09, 16#C33707D6); (* 26 *)
	c := MD5_AUX(2, c, d, a, b, X[03], 14, 16#F4D50D87); (* 27 *)
	b := MD5_AUX(2, b, c, d, a, X[08], 20, 16#455A14ED); (* 28 *)
	a := MD5_AUX(2, a, b, c, d, X[13], 05, 16#A9E3E905); (* 29 *)
	d := MD5_AUX(2, d, a, b, c, X[02], 09, 16#FCEFA3F8); (* 30 *)
	c := MD5_AUX(2, c, d, a, b, X[07], 14, 16#676F02D9); (* 31 *)
	b := MD5_AUX(2, b, c, d, a, X[12], 20, 16#8D2A4C8A); (* 32 *)

	a := MD5_AUX(3, a, b, c, d, X[05], 04, 16#FFFA3942); (* 33 *)
	d := MD5_AUX(3, d, a, b, c, X[08], 11, 16#8771F681); (* 34 *)
	c := MD5_AUX(3, c, d, a, b, X[11], 16, 16#6D9D6122); (* 35 *)
	b := MD5_AUX(3, b, c, d, a, X[14], 23, 16#FDE5380C); (* 36 *)
	a := MD5_AUX(3, a, b, c, d, X[01], 04, 16#A4BEEA44); (* 37 *)
	d := MD5_AUX(3, d, a, b, c, X[04], 11, 16#4BDECFA9); (* 38 *)
	c := MD5_AUX(3, c, d, a, b, X[07], 16, 16#F6BB4B60); (* 39 *)
	b := MD5_AUX(3, b, c, d, a, X[10], 23, 16#BEBFBC70); (* 40 *)
	a := MD5_AUX(3, a, b, c, d, X[13], 04, 16#289B7EC6); (* 41 *)
	d := MD5_AUX(3, d, a, b, c, X[00], 11, 16#EAA127FA); (* 42 *)
	c := MD5_AUX(3, c, d, a, b, X[03], 16, 16#D4EF3085); (* 43 *)
	b := MD5_AUX(3, b, c, d, a, X[06], 23, 16#04881D05); (* 44 *)
	a := MD5_AUX(3, a, b, c, d, X[09], 04, 16#D9D4D039); (* 45 *)
	d := MD5_AUX(3, d, a, b, c, X[12], 11, 16#E6DB99E5); (* 46 *)
	c := MD5_AUX(3, c, d, a, b, X[15], 16, 16#1FA27CF8); (* 47 *)
	b := MD5_AUX(3, b, c, d, a, X[02], 23, 16#C4AC5665); (* 48 *)

	a := MD5_AUX(4, a, b, c, d, X[00], 06, 16#F4292244); (* 49 *)
	d := MD5_AUX(4, d, a, b, c, X[07], 10, 16#432AFF97); (* 50 *)
	c := MD5_AUX(4, c, d, a, b, X[14], 15, 16#AB9423A7); (* 51 *)
	b := MD5_AUX(4, b, c, d, a, X[05], 21, 16#FC93A039); (* 52 *)
	a := MD5_AUX(4, a, b, c, d, X[12], 06, 16#655B59C3); (* 53 *)
	d := MD5_AUX(4, d, a, b, c, X[03], 10, 16#8F0CCC92); (* 54 *)
	c := MD5_AUX(4, c, d, a, b, X[10], 15, 16#FFEFF47D); (* 55 *)
	b := MD5_AUX(4, b, c, d, a, X[01], 21, 16#85845DD1); (* 56 *)
	a := MD5_AUX(4, a, b, c, d, X[08], 06, 16#6FA87E4F); (* 57 *)
	d := MD5_AUX(4, d, a, b, c, X[15], 10, 16#FE2CE6E0); (* 58 *)
	c := MD5_AUX(4, c, d, a, b, X[06], 15, 16#A3014314); (* 59 *)
	b := MD5_AUX(4, b, c, d, a, X[13], 21, 16#4E0811A1); (* 60 *)
	a := MD5_AUX(4, a, b, c, d, X[04], 06, 16#F7537E82); (* 61 *)
	d := MD5_AUX(4, d, a, b, c, X[11], 10, 16#BD3AF235); (* 62 *)
	c := MD5_AUX(4, c, d, a, b, X[02], 15, 16#2AD7D2BB); (* 63 *)
	b := MD5_AUX(4, b, c, d, a, X[09], 21, 16#EB86D391); (* 64 *)

	hash[0] := hash[0] + a;
	hash[1] := hash[1] + b;
	hash[2] := hash[2] + c;
	hash[3] := hash[3] + d;

END_CASE;

IF MODE = 3 THEN
	z := 0;
	FOR n := 0 TO 3 DO (* convert from little-endian to big-endian format and DWORD to BYTE array *)
		FOR n1 := 0 TO 3 DO
			MD5[z] := DWORD_TO_BYTE(hash[n]);
			hash[n] := ROR(hash[n],8);
			z := z + 1;
		END_FOR;
	END_FOR;
END_IF;
END_FUNCTION_BLOCK

// Commented out for beedance: it computes with pointers as addresses (pt := pt + 1); beedance references (REF_TO) have no arithmetic.
// FUNCTION MD5_TO_STRH : STRING(32)
// VAR_INPUT
// 	MD5 : ARRAY [0..15] OF BYTE;
// END_VAR
// VAR
// 	i : INT;
// 	tmp : BYTE;
// 	pt : REF_TO BYTE;
// END_VAR
// pt := REF(MD5_TO_STRH); (* read output adress to pointer *)
//
// FOR i := 0 TO 15 DO; (* write the 8 hex characters backwards *)
// 	tmp := SHR(MD5[i],4);
// 	PT^ := tmp + SEL(tmp <= 9,87,48);
// 	pt := pt + 1; (* decrement the pointer *)
// 	tmp := MD5[i] AND 2#1111;
// 	PT^ := tmp + SEL(tmp <= 9,87,48);
// 	pt := pt + 1; (* decrement the pointer *)
// END_FOR;
// pt^:= 0; (* write the closing byte for the string *)
// END_FUNCTION

FUNCTION_BLOCK MOON_PHASE
VAR_INPUT
	XDT : DT;
	SCALE : BYTE := 12;
	UPDATE : TIME := T#1h;
END_VAR
VAR_OUTPUT
	PHASE : BYTE;
END_VAR
VAR
	x : UDINT;
	last_dt : DT;
END_VAR

IF XDT - last_dt > UPDATE THEN
	x := (DT_TO_UDINT(XDT) - 603240) MOD 2551392;
	PHASE := UDINT_TO_BYTE(SCALE * x / 2551392) ;
	last_dt := XDT;
END_IF;
END_FUNCTION_BLOCK

// Commented out for beedance: it uses CODE, which is commented out.
// FUNCTION_BLOCK MYSQL_AUTH
// VAR_IN_OUT
// 	RUN : BOOL;
// 	PASSWORD : STRING(64);
// 	MESSAGE : ARRAY [0..19] OF BYTE;
// 	SCRAMBLE : ARRAY [0..19] OF BYTE;
// END_VAR
// VAR
// 	SHA1_STREAM : SHA1_STREAM;
// 	buf : ARRAY [0..63] OF BYTE;
// 	sha_mode : INT;
// 	step : INT;
// 	size : UDINT;
// 	pos : UDINT;
// 	i : INT;
// 	i2: INT;
// 	scramble1 : ARRAY [0..19] OF BYTE;
// 	scramble2 : ARRAY [0..19] OF BYTE;
// END_VAR
//
// IF NOT RUN THEN RETURN; END_IF;
// CASE step OF
//
// 0:	CASE sha_mode OF
// 	0:	sha_mode := 1; (* initialization *)
// 		size := INT_TO_UDINT(LEN(PASSWORD));
// 		i2 := UDINT_TO_INT(size) - 1;
// 		FOR i := 0 TO 63 DO
// 			IF i <= i2 THEN
// 				buf[i] := CODE(STR:=PASSWORD,POS:=i+1);
// 			ELSE
// 				buf[i] := BYTE#0;
// 			END_IF;
// 		END_FOR;
//
// 	3:	scramble1 := SCRAMBLE;
// 		sha_mode := 1; (* initialization *)
// 		size := UDINT#20;
// 		FOR i := 0 TO 19 DO
// 			buf[i] := scramble1[i];
// 		END_FOR;
// 		step := 10;
// 	END_CASE;
//
// 10:	IF sha_mode = 3 THEN
// 		sha_mode := 1; (* initialization *)
// 		scramble2 := SCRAMBLE;
// 		size := UDINT#40;
// 		FOR i := 0 TO 19 DO
// 			buf[i] := message[i];
// 			buf[i+20] := scramble2[i];
// 		END_FOR;
// 		step :=20;
// 	END_IF;
//
// 20:	IF sha_mode = 3 THEN
// 		sha_mode := 0; (* Stop *)
// 		FOR i:= 0 TO 19 DO
// 			SCRAMBLE[i] := SCRAMBLE[i] XOR scramble1[i];
// 		END_FOR;
// 		step :=0;
// 		RUN := FALSE;
// 	END_IF;
// END_CASE;
//
// SHA1_STREAM(SIZE:=size, MODE:=sha_mode, BUF:=buf, SHA1:=SCRAMBLE, POS=>pos);
// END_FUNCTION_BLOCK

// Commented out for beedance: it uses CODE, which is commented out.
// FUNCTION_BLOCK MYSQL_CONTROL
// VAR_IN_OUT
// 	COM : MYSQL_COM;
// 	INFO : MYSQL_INFO;
// END_VAR
// VAR_OUTPUT
// END_VAR
// VAR
// 	IP_C : IP_C;
// 	URL_DATA : url;
// 	DNS_CLIENT : DNS_CLIENT;
// 	IPC : IP_CONTROL;
//
// 	step : INT;
// 	snd_step : INT;
// 	TON_WAIT : TON;
// 	last_step : INT;
// 	idx1 : INT;
// 	idx2 : INT;
// 	idx3 : INT;
// 	dw_tmp : DWORD;
// 	timeout1 : TIME;
// 	timeout2 : TIME;
// 	ip_c_red_disable : BOOL;
// 	auth_password : STRING(64);
// 	auth_run : BOOL;
// 	MYSQL_AUTH : MYSQL_AUTH;
// 	scramble1_buffer : ARRAY [0..19] OF BYTE;
// 	scramble2_buffer : ARRAY [0..19] OF BYTE;
// 	charset_number : BYTE := 16#08;
// 	max_packet_size : DWORD := 1024;
// 	client_flags : DWORD := 16#0003_8601;
//
// 	(*
// 	LOG_MSG : LOG_MSG;
// 	_debug_enable : BOOL := TRUE;
// 	*)
//
// END_VAR
//
// CASE step OF
//
// 00:	IF COM.SQL_CON THEN
// 		timeout1 := MAX(T#10s,COM.TIMEOUT);
// 		timeout2 := timeout1 + T#1s;
// 		INFO.SQL_ERROR := '';
// 		COM.ERROR_C := DWORD#0;
// 		COM.ERROR_T := BYTE#0;
// 		URL_DATA := STRING_TO_URL(STR:=COM.SQL_URL,DEFAULT_PROTOCOL:='',DEFAULT_PATH:='/');
// 		step := 10;
// 	END_IF;
//
// 10:	IF DNS_CLIENT.DONE THEN
// 		step := 20;
// 	ELSIF DNS_CLIENT.ERROR <> DWORD#0 THEN
// 		COM.ERROR_C := DNS_CLIENT.ERROR;
// 		COM.ERROR_T := BYTE#1;
// 		step := 980;
// 	END_IF;
//
// 20:	(* set up MySQL control channel *)
// 	IF URL_DATA.PORT = WORD#0 THEN
// 		URL_DATA.PORT := WORD#3306; (* default port *)
// 	END_IF;
// 	IP_C.C_PORT := URL_DATA.PORT; (* enter port number *)
//   	IP_C.C_IP := DNS_CLIENT.IP4; (* enter IP *)
//   	IP_C.C_MODE := BYTE#0; (* Mode: TCP+ACTIV+PORT *)
//   	IP_C.TIME_RESET := TRUE; (* reset timeout monitoring *)
//   	IP_C.C_ENABLE := TRUE; (* enable connection setup *)
//   	IP_C.R_OBSERVE := TRUE; (* receive monitoring *)
// 	COM.R_BUF.SIZE := UINT#0;
// 	COM.SQL_RCV_STATE := BYTE#0;
// 	step := 30;
//
// 30:	IF COM.SQL_RCV_STATE = BYTE#1 THEN
// 		INFO.SERVER_PROTOCOL_VERSION := COM.R_BUF.BUFFER[4];
//
// 		(* search end marker of string server_version *)
// 		idx2 := UINT_TO_INT(COM.R_BUF.SIZE) - 1;
// 		FOR idx1 := 5 TO idx2 DO
// 			IF COM.R_BUF.BUFFER[idx1] = BYTE#0 THEN EXIT; END_IF;
// 		END_FOR;
// 		idx1 := idx1 + 5; (* skip termination and thread id *)
//
// 		FOR idx2:=0 TO 7 DO	(* Byte 0-7 *)
// 			scramble1_buffer[idx2] := COM.R_BUF.BUFFER[idx1];
// 			idx1 := idx1 + 1;
// 		END_FOR;
// 		idx1 := idx1 + 1;
// 		idx2 := idx1 + 1;
// 		INFO.SERVER_CAPABILITIES := WORD_OF_BYTE(COM.R_BUF.BUFFER[idx2], COM.R_BUF.BUFFER[idx1]);
// 		idx1 := idx1 + 2;
// 		INFO.SERVER_LANGUAGE := COM.R_BUF.BUFFER[idx1];
// 		idx1 := idx1 + 1;
// 		idx2 := idx1 + 1;
// 		INFO.SERVER_STATUS := WORD_OF_BYTE(COM.R_BUF.BUFFER[idx2], COM.R_BUF.BUFFER[idx1]);
// 		idx1 := idx1 + 15;
//
// 		FOR idx2:=8 TO 19 DO	(* Byte 8-19 *)
// 			scramble1_buffer[idx2] := COM.R_BUF.BUFFER[idx1];
// 			idx1 := idx1 + 1;
// 		END_FOR;
//
// 		IF INFO.SERVER_PROTOCOL_VERSION < BYTE#10 THEN  (* Error: protocol version too low *)
// 			COM.ERROR_T := BYTE#2;
// 			COM.ERROR_C := DWORD#1;
// 			step := 980;
// 		ELSIF URL_DATA.PASSWORD = '' THEN
// 			step := 50;
// 		ELSE
// 			auth_password := URL_DATA.PASSWORD;
// 			auth_run := TRUE;
// 			step := 40;
// 		END_IF;
// 	END_IF;
//
// 40:	MYSQL_AUTH(RUN:= auth_run,PASSWORD:= auth_password ,MESSAGE:= scramble1_buffer,SCRAMBLE:= scramble2_buffer);
// 	IF NOT auth_run THEN
// 		step := 50;
// 	END_IF;
//
// 50: (* Client Authentication Packet *)
// 	(* bytes 0-3 are entered later *)
// 	COM.S_BUF.BUFFER[04] := BYTE_OF_DWORD(client_flags, BYTE#0); (* client_flags *)
// 	COM.S_BUF.BUFFER[05] := BYTE_OF_DWORD(client_flags, BYTE#1);
// 	COM.S_BUF.BUFFER[06] := BYTE_OF_DWORD(client_flags, BYTE#2);
// 	COM.S_BUF.BUFFER[07] := BYTE_OF_DWORD(client_flags, BYTE#3);
// 	COM.S_BUF.BUFFER[08] := BYTE_OF_DWORD(max_packet_size, BYTE#0); (* max_packet_size *)
// 	COM.S_BUF.BUFFER[09] := BYTE_OF_DWORD(max_packet_size, BYTE#1);
// 	COM.S_BUF.BUFFER[10] := BYTE_OF_DWORD(max_packet_size, BYTE#2);
// 	COM.S_BUF.BUFFER[11] := BYTE_OF_DWORD(max_packet_size, BYTE#3);
// 	COM.S_BUF.BUFFER[12] := charset_number; (* charset_number *)
// 	FOR idx1 := 13 TO 35 DO (* 23 bytes filler always 0x00.. *)
// 		COM.S_BUF.BUFFER[idx1] := BYTE#0;
// 	END_FOR;
// 	idx3 := LEN(URL_DATA.USER);
// 	FOR idx2 :=1 TO idx3 DO
// 		COM.S_BUF.BUFFER[idx1] := CODE(URL_DATA.USER, idx2);
// 		idx1 := idx1 + 1;
// 	END_FOR;
// 	COM.S_BUF.BUFFER[idx1] := BYTE#0; (* enter string termination *)
// 	idx1 := idx1 + 1;
// 	IF LEN(URL_DATA.PASSWORD) = 0 THEN
// 		COM.S_BUF.BUFFER[idx1] := BYTE#0; (* scramble_buff length *)
// 	ELSE
// 		COM.S_BUF.BUFFER[idx1] := BYTE#20; (* scramble_buff length *)
// 		FOR idx2 :=0 TO 19 DO
// 			idx1 := idx1 + 1;
// 			COM.S_BUF.BUFFER[idx1] := scramble2_buffer[idx2];
// 		END_FOR;
// 	END_IF;
// 	COM.S_BUF.SIZE  := INT_TO_UINT(idx1 + 1); (* enter send length *)
//
// 	step := 60;
//
// 60:	IF COM.SQL_RCV_STATE = BYTE#1 THEN
// 		INFO.SQL_CONNECTED := TRUE;
// 		step := 300;
// 	END_IF;
//
// (* ================================================== *)
//
// 300:	step := SEL(COM.SQL_CON,700,310); (* step selection *)
//
// 310:	step := 300; (* dummy step *)
//
// (* ================================================== *)
//
// 700: (* COM_QUIT *)
// 	COM.S_BUF.BUFFER[04] := BYTE#1; (* 0x01 COM_QUIT mysql_close *)
// 	COM.S_BUF.SIZE := UINT#5; (* enter send length *)
// 	COM.SQL_PACKET_NO := BYTE#255;
// 	ip_c_red_disable := TRUE;
// 	step := 710;
//
// 710:	IF IP_C.C_STATE = BYTE#0 THEN (* connection closed by SQL server? *)
// 		step := 980;
// 	END_IF;
//
// (* ================================================== *)
//
// 980:IP_C.C_ENABLE := FALSE; (* close MYSQL control channel *)
// 	ip_c_red_disable := FALSE;
// 	INFO.SQL_CONNECTED := FALSE;
// 	COM.SQL_CON := FALSE;
// 	COM.S_BUF.SIZE := UINT#0;
// 	COM.R_BUF.SIZE := UINT#0;
// 	snd_step := 0;
// 	step := 990;
// 	(*####################  DEBUG-MESSAGE  ###################################*)
// 	(*IF _debug_enable THEN
// 		LOG_CL.NEW_MSG := 'QUIT: ERROR CODE >~1< TYPE >~2<';
// 		LOG_CL.PRINTF[1] := DWORD_TO_STRH(COM.ERROR_C);
// 		LOG_CL.PRINTF[2] := BYTE_TO_STRING(COM.ERROR_T);
// 		LOG_MSG();
// 	END_IF;*)
// 	(*########################################################################*)
//
// 990:IF IP_C.C_STATE = BYTE#0 THEN
// 		step := 0;
// 	END_IF;
//
// END_CASE;
//
// (* ++++++++++++++++++++++++++++++++++++++++++++++++++++++++++ *)
//
// IF step >= 30 THEN
// 	IF COM.R_BUF.SIZE >= UINT#3 AND COM.SQL_RCV_STATE = BYTE#0 THEN (* data received? *)
// 		IF DWORD_TO_UINT(DWORD_OF_BYTE(BYTE#0, COM.R_BUF.BUFFER[2], COM.R_BUF.BUFFER[1], COM.R_BUF.BUFFER[0])) + UINT#4 = COM.R_BUF.SIZE THEN
// 			COM.SQL_PACKET_NO := COM.R_BUF.BUFFER[3];
// 			IF COM.R_BUF.BUFFER[4] = BYTE#16#FF THEN
// 				idx2 := 13; (* error string - first character *)
// 				idx3 := UINT_TO_INT(COM.R_BUF.SIZE) - 1; (* error string - last character *)
// 				FOR idx1 := idx2 TO idx3 DO (* replace all ' with ´ *)
// 					IF COM.R_BUF.BUFFER[idx1] = BYTE#39 THEN
// 						COM.R_BUF.BUFFER[idx1] := BYTE#96;
// 					END_IF;
// 				END_FOR;
// 				INFO.SQL_ERROR := BUFFER_TO_STRING(PT:=REF(COM.R_BUF.BUFFER),SIZE:=COM.R_BUF.SIZE,START:=INT_TO_UINT(idx2),STOP:=INT_TO_UINT(idx3));
// 				COM.ERROR_T := BYTE#3;
// 				COM.ERROR_C := DWORD_OF_BYTE(BYTE#0,BYTE#0,COM.R_BUF.BUFFER[6], COM.R_BUF.BUFFER[5]);
// 				COM.SQL_RCV_STATE := BYTE#2;
// 				COM.R_BUF.SIZE := UINT#0; (* reset receive buffer after error *)
// 				step := 980;
// 			ELSE
// 				COM.SQL_RCV_STATE := BYTE#1;
// 				IP_C.R_OBSERVE := FALSE;
//
// 				(*####################  DEBUG-MESSAGE  ###################################*)
// 				(*IF _debug_enable THEN
// 					LOG_CL.NEW_MSG := 'RCV: size >~1<';
// 					LOG_CL.PRINTF[1] := UINT_TO_STRING(COM.R_BUF.SIZE);
// 					LOG_MSG();
// 				END_IF;*)
// 				(*########################################################################*)
// 			END_IF;
// 		END_IF;
// 	END_IF;
// END_IF;
//
// (* automatic data sending *)
//
// CASE snd_step OF
//
// 00:	IF step >= 20 AND COM.S_BUF.SIZE > UINT#0 THEN
// 		dw_tmp := UINT_TO_DWORD(COM.S_BUF.SIZE - UINT#4); (* packet_length *)
// 		COM.S_BUF.BUFFER[0] := BYTE_OF_DWORD(dw_tmp, BYTE#0);
// 		COM.S_BUF.BUFFER[1] := BYTE_OF_DWORD(dw_tmp, BYTE#1);
// 		COM.S_BUF.BUFFER[2] := 0;
// 		COM.SQL_PACKET_NO := COM.SQL_PACKET_NO + 1;
// 		COM.S_BUF.BUFFER[3] := COM.SQL_PACKET_NO;
//
// 		IP_C.R_OBSERVE := TRUE;
// 		COM.R_BUF.SIZE := UINT#0; (* reset receive buffer *)
// 		COM.SQL_RCV_STATE := BYTE#0;
//
// 	        (*####################  DEBUG-MESSAGE  ###################################*)
// 	        (*IF _debug_enable THEN
// 	          LOG_CL.NEW_MSG := 'SND: size >~1<';
// 	          LOG_CL.PRINTF[1] := UINT_TO_STRING(COM.S_BUF.SIZE);
// 	          LOG_MSG();
// 	        END_IF;*)
// 	        (*########################################################################*)
//
// 		snd_step := 10;
// 	END_IF;
//
// 10:	IF COM.S_BUF.SIZE = UINT#0 THEN (* wait until all data is sent *)
// 		snd_step := 0;
// 	END_IF;
//
// END_CASE;
//
// (* global error handling for main routine *)
// IF COM.ERROR_T = BYTE#0 AND step > 20 THEN (* no error stored yet and main routine active *)
// 	IF IP_C.ERROR > DWORD#0 AND IP_C.C_ENABLE AND NOT IP_C.TIME_RESET THEN  (* IP Control *)
// 		IF ip_c_red_disable = FALSE OR IP_C.ERROR <> DWORD#16#FD000000 THEN
// 			COM.ERROR_C := IP_C.ERROR;
// 			COM.ERROR_T := BYTE#2;
// 			step := 980;
// 		END_IF;
// 	END_IF;
// END_IF;
//
// IF TON_WAIT.Q THEN (* sequence fault - step chain *)
// 	COM.ERROR_C := INT_TO_DWORD(step); (* enter current step *)
// 	COM.ERROR_T := BYTE#5;
// 	step := 980;
// END_IF;
//
// (* ######################################################## *)
//
// DNS_CLIENT(IP_C:=IP_C, S_BUF:=COM.S_BUF, R_BUF:=COM.R_BUF, DOMAIN:=URL_DATA.DOMAIN, IP4_DNS:= COM.DNS_IP4, ACTIVATE:=step=10); (* DNS-Client *)
// IPC(IP:= DWORD#0, PORT:= WORD#0 , TIME_OUT:= timeout1, IP_C:= IP_C, S_BUF:= COM.S_BUF, R_BUF:= COM.R_BUF); (* MYSQL control channel *)
//
// TON_WAIT(IN:=step = last_step AND step > 0,PT:=timeout2);
// last_step := step;
// END_FUNCTION_BLOCK

FUNCTION_BLOCK NET_VAR_BOOL8
VAR_IN_OUT
	X : NET_VAR_DATA;
END_VAR
VAR_INPUT
	IN1 : BOOL;
	IN2 : BOOL;
	IN3 : BOOL;
	IN4 : BOOL;
	IN5 : BOOL;
	IN6 : BOOL;
	IN7 : BOOL;
	IN8 : BOOL;
END_VAR
VAR_OUTPUT
	OUT1 : BOOL;
	OUT2 : BOOL;
	OUT3 : BOOL;
	OUT4 : BOOL;
	OUT5 : BOOL;
	OUT6 : BOOL;
	OUT7 : BOOL;
	OUT8 : BOOL;
	ID : BYTE;
END_VAR
VAR
	init : BOOL;
	index : INT;
	index2 : INT;
	BYTE_TO_BITS : BYTE_TO_BITS;
END_VAR

IF NOT init THEN
	init := TRUE;
	X.ID_MAX := X.ID_MAX + USINT#1;
	ID := USINT_TO_BYTE(X.ID_MAX);
END_IF;

IF X.STATE > BYTE#0 AND X.ERROR_ID = BYTE#0 THEN
	index := X.index; (* PCWORX Workaround *)
	IF INT_TO_UINT(index + 3) > X.BUF_SIZE THEN
		X.ERROR_ID := ID;
	ELSE
		IF X.STATE = BYTE#1 THEN (* write data *)
			X.S_BUF.BUFFER[index] := ID; (* ID *)
			index := index + 1;
			X.S_BUF.BUFFER[index] := BYTE#4; (* TYPE BOOL8 *)
			index := index + 1;
			X.S_BUF.BUFFER[index] := BYTE_OF_BIT(IN1,IN2,IN3,IN4,IN5,IN6,IN7,IN8);
			index := index + 1;

		ELSIF X.STATE = BYTE#2 THEN (* read data *)
			index2 := index + 1; (* PCWORX Workaround *)
			IF X.R_BUF.BUFFER[index] <> ID OR X.R_BUF.BUFFER[index2] <> BYTE#4 THEN
				X.ERROR_ID := ID;
			ELSE
				index := index + 2;
				BYTE_TO_BITS(IN:=X.R_BUF.BUFFER[index]);
				OUT1 := BYTE_TO_BITS.B0;
				OUT2 := BYTE_TO_BITS.B1;
				OUT3 := BYTE_TO_BITS.B2;
				OUT4 := BYTE_TO_BITS.B3;
				OUT5 := BYTE_TO_BITS.B4;
				OUT6 := BYTE_TO_BITS.B5;
				OUT7 := BYTE_TO_BITS.B6;
				OUT8 := BYTE_TO_BITS.B7;
				index := index + 1;
			END_IF;
		END_IF;
		X.index := index;
	END_IF;
END_IF;
END_FUNCTION_BLOCK

FUNCTION_BLOCK NET_VAR_BUFFER
VAR_IN_OUT
	BUF_IN : ARRAY[1..64] OF BYTE;
	BUF_OUT : ARRAY[1..64] OF BYTE;
	X : NET_VAR_DATA;
END_VAR
VAR_OUTPUT
	ID : BYTE;
END_VAR
VAR
	size : INT;
	init : BOOL;
	index : INT;
	index2 : INT;
END_VAR

IF NOT init THEN
	init := TRUE;
	X.ID_MAX := X.ID_MAX + USINT#1;
	ID := USINT_TO_BYTE(X.ID_MAX);
END_IF;

IF X.STATE > BYTE#0 AND X.ERROR_ID = BYTE#0 THEN
	index := X.index; (* PCWORX Workaround *)
	IF X.STATE = BYTE#1 THEN (* write data *)
		size := SIZEOF(BUF_IN);
		IF INT_TO_UINT(index + 3 + size) > X.BUF_SIZE THEN
			X.ERROR_ID := ID;
		ELSE
			X.S_BUF.BUFFER[index] := ID; (* ID *)
			index := index + 1;
			X.S_BUF.BUFFER[index] := BYTE#20; (* TYPE BUFFER *)
			index := index + 1;
			X.S_BUF.BUFFER[index] := INT_TO_BYTE(size); (* number of bytes *)
				index := index + 1;
			FOR index2 := 1 TO size DO
				X.S_BUF.BUFFER[index] := BUF_IN[index2];
				index := index + 1;
			END_FOR;
		END_IF;
	ELSIF X.STATE = BYTE#2 THEN (* read data *)
		index2 := index + 1; (* PCWORX Workaround *)
		IF X.R_BUF.BUFFER[index] <> ID OR X.R_BUF.BUFFER[index2] <> BYTE#20 THEN
			X.ERROR_ID := ID;
		ELSE
			index := index + 2;
			size := BYTE_TO_INT(X.R_BUF.BUFFER[index]);
			index := index + 1;
			FOR index2 := 1 TO size DO
				BUF_OUT[index2] := X.R_BUF.BUFFER[index];
				index := index + 1;
			END_FOR;
		END_IF;
	END_IF;
	X.index := index;
END_IF;
END_FUNCTION_BLOCK

// Commented out for beedance: beedance cannot yet tell SIZEOF(X.S_BUF.BUFFER), the size of a member of the VAR_IN_OUT X.
// FUNCTION_BLOCK NET_VAR_CONTROL
// VAR_INPUT
// 	ACTIVATE : BOOL;
// 	MASTER : BOOL;
// 	UDP : BOOL;
// 	REMOTE_IP4 : DWORD;
// 	REMOTE_PORT : WORD := 10000;
// 	SCAN_TIME : TIME := T#1s;
// 	WATCHDOG : TIME := T#2s;
// END_VAR
// VAR_OUTPUT
// 	RUN : BOOL;
// 	ERROR : DWORD;
// END_VAR
// VAR_IN_OUT
// 	X : NET_VAR_DATA;
// END_VAR
// VAR
// 	IPC : IP_CONTROL;
// 	IP_C : IP_C; (* IP_Control management structure *)
// 	step : INT;
// 	activate_last : BOOL;
// 	tscan : TON;
// 	reset : BOOL;
// END_VAR
//
// IF X.ERROR_ID > BYTE#0 THEN (* severe errors in variable assignment present  !! *)
// 	X.STATE := BYTE#0;
// 	ERROR := BYTE_TO_DWORD(X.ERROR_ID);
// 	X.ERROR_ID := BYTE#0;
// 	step := 999;
// END_IF;
//
// CASE step OF
//
// 00:	IF ACTIVATE AND NOT activate_last OR reset THEN
//
//         (*  TCP + MASTER = C_MODE 0 (TCP + ACTIVE + PORT + IP) *)
//         (*  UDP + MASTER = C_MODE 1 (UDP + ACTIVE + PORT + IP) *)
//         (*  TCP + SLAVE  = C_MODE 2 (TCP + PASSIVE + PORT + IP) *)
//         (*  UDP + SLAVE  = C_MODE 3 (UDP + PASSIVE + PORT + IP) *)
// 	IF MASTER THEN
// 		IP_C.C_MODE := BYTE#0;
// 		step := 100;
// 	ELSE
// 		IP_C.C_MODE := BYTE#2;
// 		step := 200;
// 	END_IF;
//         IF UDP THEN IP_C.C_MODE := IP_C.C_MODE OR BYTE#1; END_IF;
// 	  	IP_C.C_PORT := REMOTE_PORT; (* enter port number *)
// 	  	IP_C.C_IP := REMOTE_IP4; (* enter IP *)
// 	  	IP_C.TIME_RESET := TRUE; (* reset timeout monitoring *)
// 	  	IP_C.C_ENABLE := TRUE; (* enable connection setup *)
// 	  	IP_C.R_OBSERVE := TRUE; (* receive monitoring *)
// 		X.S_BUF.SIZE := UINT#0;
// 		X.R_BUF.SIZE := UINT#0;
// 		X.CYCLE := UDINT#0;
// 		X.ERROR_ID := BYTE#0;
// 		reset := FALSE;
// 	END_IF;
//
// (* ++++++++++++++++++++++++++++++++++++++++++++++ *)
//
// 100:IF IP_C.C_STATE > BYTE#127 THEN (* connection present *)
// 		X.STATE := BYTE#1; (* collect data *)
// 		X.BUF_SIZE := SIZEOF(X.S_BUF.BUFFER);
// 		X.S_BUF.BUFFER[0] := UDINT_TO_BYTE(X.CYCLE);
// 		X.INDEX := 1;
// 		step := 110;
// 	END_IF;
//
// 110:X.STATE := BYTE#0;
// 	X.S_BUF.SIZE := INT_TO_UINT(X.INDEX); (* enter data length *)
// 	step := 120;
//
// 120:IF X.S_BUF.SIZE = UINT#0 AND X.R_BUF.SIZE >= UINT#1 THEN (* check length of received data *)
// 		X.STATE := BYTE#2; (* output data *)
// 		X.BUF_SIZE := X.R_BUF.SIZE;
// 		X.INDEX := 1;
// 		X.ERROR_ID := BYTE#0;
// 		X.CYCLE := X.CYCLE + UDINT#1;
// 		ERROR := DWORD#0; (* clear last error code after a successful cycle *)
// 		RUN := TRUE;
// 		step := 130;
// 	END_IF;
//
// 130:X.STATE := BYTE#0;
// 	X.R_BUF.SIZE := UINT#0;
// 	IF NOT ACTIVATE THEN
// 		step := 999; (* exit *)
// 	ELSIF tscan.Q THEN
// 		step := 100;
// 	END_IF;
//
// (* ++++++++++++++++++++++++++++++++++++++++++++++ *)
//
// 200:IF X.R_BUF.SIZE >= UINT#1 THEN
// 		X.STATE := BYTE#2; (* output data *)
// 		X.BUF_SIZE := X.R_BUF.SIZE;
// 		X.INDEX := 1;
// 		step := 210;
// 	END_IF;
//
// 210:X.STATE := BYTE#1; (* collect data *)
// 	X.BUF_SIZE := SIZEOF(X.R_BUF.BUFFER);;
// 	X.S_BUF.BUFFER[0] := X.R_BUF.BUFFER[0]; (* take cycle *)
// 	X.INDEX := 1;
// 	X.R_BUF.SIZE := UINT#0;
// 	step := 220;
//
// 220:X.STATE := BYTE#0;
// 	X.S_BUF.SIZE := INT_TO_UINT(X.INDEX); (* enter data length *)
// 	step := 230;
//
// 230:IF X.S_BUF.SIZE = UINT#0 THEN
// 		ERROR := DWORD#0; (* clear last error code after a successful cycle *)
// 		RUN := TRUE;
// 		IF NOT ACTIVATE THEN
// 			step := 999; (* exit *)
// 		ELSE
// 			step := 200;
// 		END_IF;
// 	END_IF;
//
// 999:IP_C.C_ENABLE := FALSE; (* exit *)
// 	RUN := FALSE;
// 	step := 0;
//
// END_CASE;
//
// (* ++++++++++++++++++++++++++++++++++++++++++++++ *)
//
// IPC(IP:= DWORD#0, PORT:= WORD#0 , TIME_OUT:= WATCHDOG, IP_C:= IP_C, S_BUF:= X.S_BUF, R_BUF:= X.R_BUF);
//
// IF IP_C.ERROR > DWORD#0 THEN
// 	ERROR := IP_C.ERROR;
// 	RUN := FALSE;
// 	reset := TRUE;
// 	step := 0;
// END_IF;
//
// ACTIVATE_LAST := ACTIVATE; (* save last status for edge detection *)
// tscan(IN:= step <> 110 ,PT:=SCAN_TIME);
// END_FUNCTION_BLOCK

FUNCTION_BLOCK NET_VAR_DWORD8
VAR_IN_OUT
	X : NET_VAR_DATA;
END_VAR
VAR_INPUT
	IN1 : DWORD;
	IN2 : DWORD;
	IN3 : DWORD;
	IN4 : DWORD;
	IN5 : DWORD;
	IN6 : DWORD;
	IN7 : DWORD;
	IN8 : DWORD;
END_VAR
VAR_OUTPUT
	OUT1 : DWORD;
	OUT2 : DWORD;
	OUT3 : DWORD;
	OUT4 : DWORD;
	OUT5 : DWORD;
	OUT6 : DWORD;
	OUT7 : DWORD;
	OUT8 : DWORD;
	ID : BYTE;
END_VAR
VAR
	init : BOOL;
	i : INT;
	i2 : INT;
	index : INT;
	index2 : INT;
	ra : ARRAY[1..8] OF DWORD;
END_VAR

IF NOT init THEN
	init := TRUE;
	X.ID_MAX := X.ID_MAX + USINT#1;
	ID := USINT_TO_BYTE(X.ID_MAX);
END_IF;

IF X.STATE > BYTE#0 AND X.ERROR_ID = BYTE#0 THEN
	index := X.index; (* PCWORX Workaround *)
	IF INT_TO_UINT(index + 34) > X.BUF_SIZE THEN  (* ID (1) + TYPE (1) + 8 x DWORD (4) *)
		X.ERROR_ID := ID;
	ELSE
		IF X.STATE = BYTE#1 THEN (* write data *)
			ra[1] := IN1;
			ra[2] := IN2;
			ra[3] := IN3;
			ra[4] := IN4;
			ra[5] := IN5;
			ra[6] := IN6;
			ra[7] := IN7;
			ra[8] := IN8;
			X.S_BUF.BUFFER[index] := ID; (* ID *)
			index := index + 1;
			X.S_BUF.BUFFER[index] := BYTE#13; (* TYPE DWORD8 *)
			index := index + 1;
			FOR i2 := 1 TO 8 DO;
				FOR i := 1 TO 4 DO;
					X.S_BUF.BUFFER[index] := DWORD_TO_BYTE(ra[i2]);
					ra[i2] := ROR(ra[i2],8);
					index := index + 1;
				END_FOR;
			END_FOR;
